// TIA Portal project "Project3" (V17)

(* hardware
DEVICE "S7-1200 station_1"  S7-1200 Station
   slot 0: "Rack_0"  S7-1200 Rack  Rack  V1.0
   slot 1: "PLC_1"  CPU 1212C DC/DC/DC  6ES7 212-1AE40-0XB0  V4.2
DEVICE "HMI_1"  TP700 Comfort
   slot 0: "HMI_1"  TP700 Comfort  6AV2 124-0GC01-0AX0  17.0.0.0
   slot 1: "HMI_RT_1"  TP700 Comfort  6AV2 124-0GC01-0AX0  17.0.0.0
   slot 5: "HMI_1.IE_CP_1"  PROFINET Interface  17.0.0.0
      slot 1: "PROFINET Interface_1"  PROFINET Interface
         slot 1: "Port_1"  Port
         slot 2: "Port_2"  Port
   slot 7: "HMI_1.MPI/DP_CP_1"  MPI/DP Interface  17.0.0.0
*)

// ===== PLC "PLC_1"  CPU 1212C DC/DC/DC =====

VAR_GLOBAL   // PLC tag table "Default tag table"
   "S2" AT %I0.0 : Bool;
   "S3" AT %I0.1 : Bool;
   "S1" AT %I0.2 : Bool;
   "S4" AT %I0.3 : Bool;
   "S5" AT %I0.4 : Bool;
   "Ac" AT %Q0.0 : Bool;
   "Aż" AT %Q0.1 : Bool;
   "Az" AT %Q0.2 : Bool;
   "Bc" AT %Q0.3 : Bool;
   "Bż" AT %Q0.4 : Bool;
   "Bz" AT %Q0.5 : Bool;
   "Clock_Byte" AT %MB100 : Byte;
   "Clock_10Hz" AT %M100.0 : Bool;
   "Clock_5Hz" AT %M100.1 : Bool;
   "Clock_2.5Hz" AT %M100.2 : Bool;
   "Clock_2Hz" AT %M100.3 : Bool;
   "Clock_1.25Hz" AT %M100.4 : Bool;
   "Clock_1Hz" AT %M100.5 : Bool;
   "Clock_0.625Hz" AT %M100.6 : Bool;
   "Clock_0.5Hz" AT %M100.7 : Bool;
   "Start_HMI" AT %M0.0 : Bool;
   "Stop_HMI" AT %M0.1 : Bool;
   "ŻądaniePrzejazdu_HMI" AT %M0.2 : Bool;
   "TrybNocny_HMI" AT %M0.3 : Bool;
   "ResetAwarii_HMI" AT %M0.4 : Bool;
   "Auto/Manual_przycisk" AT %M0.5 : Bool;
   "Ac_HMI" AT %M0.6 : Bool;
   "Aż_HMI" AT %M0.7 : Bool;
   "Az_HMI" AT %M1.0 : Bool;
   "Bc_HMI" AT %M1.1 : Bool;
   "Bż_HMI" AT %M1.2 : Bool;
   "Bz_HMI" AT %M1.3 : Bool;
END_VAR

DATA_BLOCK "Data_block_1"   // DB1
{ S7_Optimized_Access := 'TRUE' }
VERSION : 0.1
   VAR
      ImpulsS4 : Bool;
      TrybNocny : Bool;
      PamiecZboczaS4 : Bool;
      LicznikS4 : Int;
      Awaria : Bool;
      LiczbaCykli : DInt;
      LiczbaPojazdow : DInt;
      LiczbaŻądań : DInt;
      PamiecZboczaS3_2 : Bool;
      PamiecZboczaS3_1 : Bool;
      PamiecZboczaS3 : Bool;
      NumerAktualnegoKroku : Int;
      Pamięć_HMI_Az : Bool;
      Pamięć_HMI_Bz : Bool;
      Pamięć_HMI_Aż : Bool;
      Pamięć_HMI_Bż : Bool;
      Pamięć_HMI_Ac : Bool;
      Pamięć_HMI_Bc : Bool;
      Impuls_HMI_Az : Bool;
      Impuls_HMI_Bz : Bool;
      Impuls_HMI_Aż : Bool;
      Impuls_HMI_Bż : Bool;
      Impuls_HMI_Ac : Bool;
      Impuls_HMI_Bc : Bool;
      Zmiana_Kroku_Wykonana : Bool;
   END_VAR
BEGIN
END_DATA_BLOCK

// folder: System blocks/Program resources

DATA_BLOCK "IEC_Counter_0_DB"   // DB2
{ S7_Optimized_Access := 'TRUE' }
AUTHOR : Simatic
FAMILY : IEC
NAME : CNTR
VERSION : 1.0
// stored: InstanceOfName IEC_COUNTER
"IEC_COUNTER"
BEGIN
END_DATA_BLOCK

DATA_BLOCK "IEC_Timer_0_DB_1"   // DB3
{ S7_Optimized_Access := 'TRUE' }
AUTHOR : Simatic
FAMILY : IEC
NAME : IEC_TMR
VERSION : 1.0
// stored: InstanceOfName IEC_TIMER
"IEC_TIMER"
BEGIN
END_DATA_BLOCK

DATA_BLOCK "IEC_Timer_0_DB_2"   // DB4
{ S7_Optimized_Access := 'TRUE' }
AUTHOR : Simatic
FAMILY : IEC
NAME : IEC_TMR
VERSION : 1.0
// stored: InstanceOfName IEC_TIMER
"IEC_TIMER"
BEGIN
END_DATA_BLOCK

DATA_BLOCK "IEC_Timer_0_DB_3"   // DB5
{ S7_Optimized_Access := 'TRUE' }
AUTHOR : Simatic
FAMILY : IEC
NAME : IEC_TMR
VERSION : 1.0
// stored: InstanceOfName IEC_TIMER
"IEC_TIMER"
BEGIN
END_DATA_BLOCK

DATA_BLOCK "IEC_Timer_0_DB_4"   // DB6
{ S7_Optimized_Access := 'TRUE' }
AUTHOR : Simatic
FAMILY : IEC
NAME : IEC_TMR
VERSION : 1.0
// stored: InstanceOfName IEC_TIMER
"IEC_TIMER"
BEGIN
END_DATA_BLOCK

DATA_BLOCK "IEC_Timer_0_DB_5"   // DB7
{ S7_Optimized_Access := 'TRUE' }
AUTHOR : Simatic
FAMILY : IEC
NAME : IEC_TMR
VERSION : 1.0
// stored: InstanceOfName IEC_TIMER
"IEC_TIMER"
BEGIN
END_DATA_BLOCK

DATA_BLOCK "IEC_Timer_0_DB_6"   // DB8
{ S7_Optimized_Access := 'TRUE' }
AUTHOR : Simatic
FAMILY : IEC
NAME : IEC_TMR
VERSION : 1.0
// stored: InstanceOfName IEC_TIMER
"IEC_TIMER"
BEGIN
END_DATA_BLOCK

DATA_BLOCK "IEC_Timer_0_DB_7"   // DB9
{ S7_Optimized_Access := 'TRUE' }
AUTHOR : Simatic
FAMILY : IEC
NAME : IEC_TMR
VERSION : 1.0
// stored: InstanceOfName IEC_TIMER
"IEC_TIMER"
BEGIN
END_DATA_BLOCK

DATA_BLOCK "IEC_Timer_0_DB_8"   // DB10
{ S7_Optimized_Access := 'TRUE' }
AUTHOR : Simatic
FAMILY : IEC
NAME : IEC_TMR
VERSION : 1.0
// stored: InstanceOfName IEC_TIMER
"IEC_TIMER"
BEGIN
END_DATA_BLOCK

DATA_BLOCK "IEC_Counter_0_DB_1"   // DB11
{ S7_Optimized_Access := 'TRUE' }
AUTHOR : Simatic
FAMILY : IEC
NAME : CNTR
VERSION : 1.0
// stored: InstanceOfName IEC_COUNTER
"IEC_COUNTER"
BEGIN
END_DATA_BLOCK

DATA_BLOCK "IEC_Timer_0_DB"   // DB12
{ S7_Optimized_Access := 'TRUE' }
AUTHOR : Simatic
FAMILY : IEC
NAME : IEC_TMR
VERSION : 1.0
// stored: InstanceOfName IEC_TIMER
"IEC_TIMER"
BEGIN
END_DATA_BLOCK

DATA_BLOCK "IEC_Counter_0_DB_5"   // DB13
{ S7_Optimized_Access := 'TRUE' }
AUTHOR : Simatic
FAMILY : IEC
NAME : CNTR
VERSION : 1.0
// stored: InstanceOfName IEC_COUNTER
"IEC_COUNTER"
BEGIN
END_DATA_BLOCK

DATA_BLOCK "IEC_Timer_0_DB_9"   // DB14
{ S7_Optimized_Access := 'TRUE' }
AUTHOR : Simatic
FAMILY : IEC
NAME : IEC_TMR
VERSION : 1.0
// stored: InstanceOfName IEC_TIMER
"IEC_TIMER"
BEGIN
END_DATA_BLOCK

DATA_BLOCK "IEC_Counter_0_DB_4"   // DB15
{ S7_Optimized_Access := 'TRUE' }
AUTHOR : Simatic
FAMILY : IEC
NAME : CNTR
VERSION : 1.0
// stored: InstanceOfName IEC_COUNTER
"IEC_COUNTER"
BEGIN
END_DATA_BLOCK

DATA_BLOCK "IEC_Timer_0_DB_13"   // DB16
{ S7_Optimized_Access := 'TRUE' }
AUTHOR : Simatic
FAMILY : IEC
NAME : IEC_TMR
VERSION : 1.0
// stored: InstanceOfName IEC_TIMER
"IEC_TIMER"
BEGIN
END_DATA_BLOCK

DATA_BLOCK "IEC_Timer_0_DB_14"   // DB17
{ S7_Optimized_Access := 'TRUE' }
AUTHOR : Simatic
FAMILY : IEC
NAME : IEC_TMR
VERSION : 1.0
// stored: InstanceOfName IEC_TIMER
"IEC_TIMER"
BEGIN
END_DATA_BLOCK

DATA_BLOCK "IEC_Timer_0_DB_15"   // DB18
{ S7_Optimized_Access := 'TRUE' }
AUTHOR : Simatic
FAMILY : IEC
NAME : IEC_TMR
VERSION : 1.0
// stored: InstanceOfName IEC_TIMER
"IEC_TIMER"
BEGIN
END_DATA_BLOCK

DATA_BLOCK "IEC_Timer_0_DB_16"   // DB19
{ S7_Optimized_Access := 'TRUE' }
AUTHOR : Simatic
FAMILY : IEC
NAME : IEC_TMR
VERSION : 1.0
// stored: InstanceOfName IEC_TIMER
"IEC_TIMER"
BEGIN
END_DATA_BLOCK

DATA_BLOCK "IEC_Timer_0_DB_17"   // DB20
{ S7_Optimized_Access := 'TRUE' }
AUTHOR : Simatic
FAMILY : IEC
NAME : IEC_TMR
VERSION : 1.0
// stored: InstanceOfName IEC_TIMER
"IEC_TIMER"
BEGIN
END_DATA_BLOCK

DATA_BLOCK "IEC_Timer_0_DB_18"   // DB21
{ S7_Optimized_Access := 'TRUE' }
AUTHOR : Simatic
FAMILY : IEC
NAME : IEC_TMR
VERSION : 1.0
// stored: InstanceOfName IEC_TIMER
"IEC_TIMER"
BEGIN
END_DATA_BLOCK

DATA_BLOCK "IEC_Timer_0_DB_10"   // DB22
{ S7_Optimized_Access := 'TRUE' }
AUTHOR : Simatic
FAMILY : IEC
NAME : IEC_TMR
VERSION : 1.0
// stored: InstanceOfName IEC_TIMER
"IEC_TIMER"
BEGIN
END_DATA_BLOCK

DATA_BLOCK "IEC_Timer_0_DB_11"   // DB23
{ S7_Optimized_Access := 'TRUE' }
AUTHOR : Simatic
FAMILY : IEC
NAME : IEC_TMR
VERSION : 1.0
// stored: InstanceOfName IEC_TIMER
"IEC_TIMER"
BEGIN
END_DATA_BLOCK

DATA_BLOCK "IEC_Timer_0_DB_12"   // DB24
{ S7_Optimized_Access := 'TRUE' }
AUTHOR : Simatic
FAMILY : IEC
NAME : IEC_TMR
VERSION : 1.0
// stored: InstanceOfName IEC_TIMER
"IEC_TIMER"
BEGIN
END_DATA_BLOCK

// folder: (top level)

ORGANIZATION_BLOCK "Main"   // OB1, LAD, ProgramCycle
TITLE = "Main Program Sweep (Cycle)"
{ S7_Optimized_Access := 'TRUE' }
VERSION : 0.1
   VAR_INPUT
      Initial_Call : Bool;   // Initial call of this OB
      Remanence : Bool;   // =True, if remanent data are available
   END_VAR
   VAR_TEMP   // added for the SCL form of the ladder/FBD networks
      _w1 : Bool;
      _w2 : Bool;
      _w3 : Bool;
      _w4 : Bool;
      _w5 : Bool;
      _w6 : Bool;
   END_VAR
BEGIN

REGION Network 1: Inicjalizacja programu
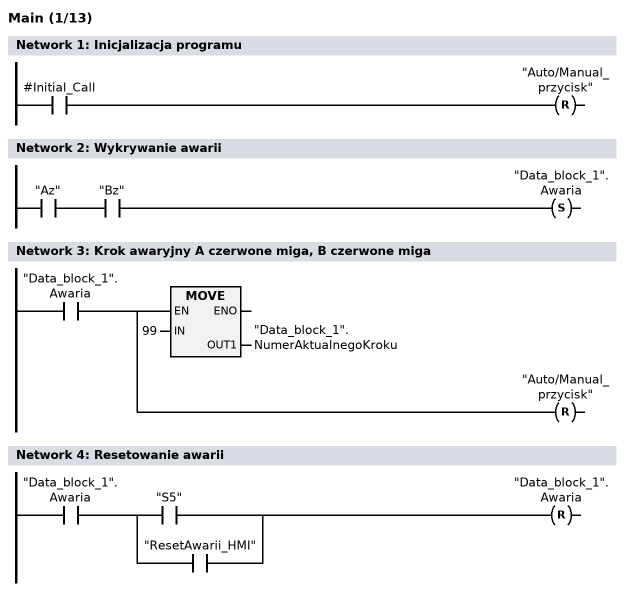
   RUNG wire#powerrail
      Contact( #Initial_Call )
      R_Coil( "Auto/Manual_przycisk" )
   END_RUNG
   // the same network as SCL:
   IF #Initial_Call THEN "Auto/Manual_przycisk" := FALSE; END_IF;
END_REGION

REGION Network 2: Wykrywanie awarii
   RUNG wire#powerrail
      Contact( "Az" )
      Contact( "Bz" )
      S_Coil( "Data_block_1".Awaria )
   END_RUNG
   // the same network as SCL:
   IF "Az" AND "Bz" THEN "Data_block_1".Awaria := TRUE; END_IF;
END_REGION

REGION Network 3: Krok awaryjny A czerwone miga, B czerwone miga
   RUNG wire#powerrail
      Contact( "Data_block_1".Awaria )
      wire#w1
      Move(in := 99, out1 => "Data_block_1".NumerAktualnegoKroku)
   END_RUNG
   RUNG wire#w1
      R_Coil( "Auto/Manual_przycisk" )
   END_RUNG
   // the same network as SCL:
   IF "Data_block_1".Awaria THEN
       "Data_block_1".NumerAktualnegoKroku := 99;
       "Auto/Manual_przycisk" := FALSE;
   END_IF;
END_REGION

REGION Network 4: Resetowanie awarii
   RUNG wire#powerrail
      Contact( "Data_block_1".Awaria )
      wire#w1
      Contact( "S5" )
      wire#w2
      R_Coil( "Data_block_1".Awaria )
   END_RUNG
   RUNG wire#w1
      Contact( "ResetAwarii_HMI" )
   END_RUNG wire#w2
   // the same network as SCL:
   IF "Data_block_1".Awaria AND ("S5" OR "ResetAwarii_HMI") THEN "Data_block_1".Awaria := FALSE; END_IF;
END_REGION

REGION Network 5: Tryb nocny
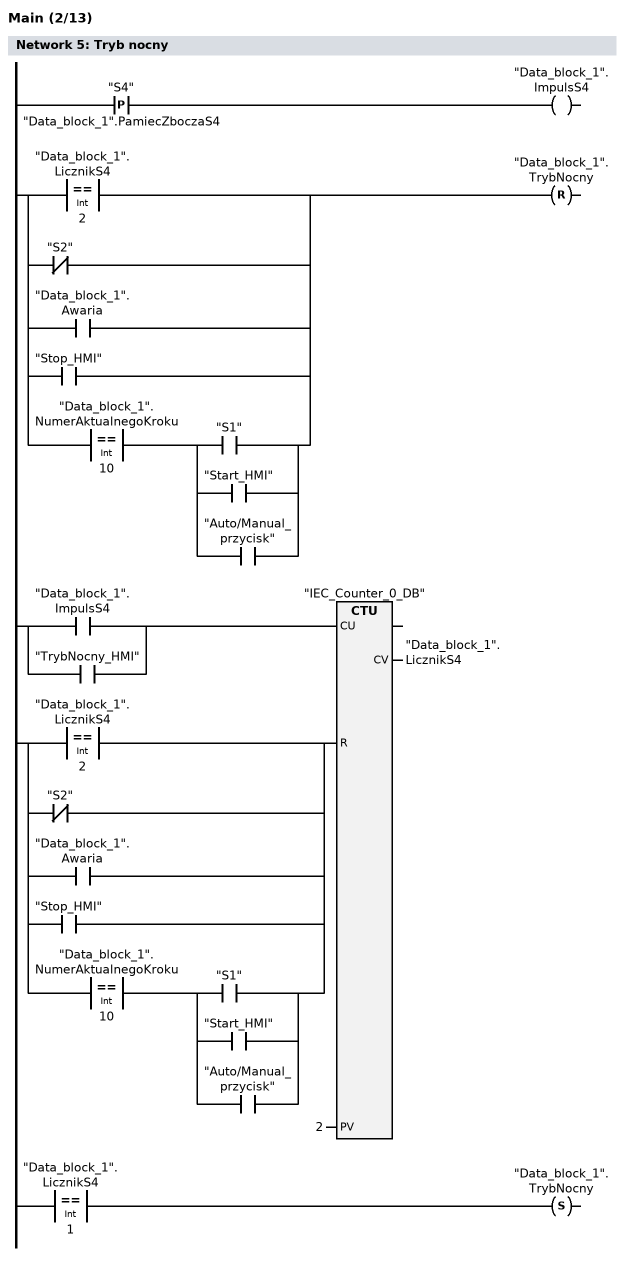
   #_w1 := "S4" AND NOT "Data_block_1".PamiecZboczaS4;   // rising edge of "S4"
   "Data_block_1".PamiecZboczaS4 := "S4";
   "Data_block_1".ImpulsS4 := #_w1;
   IF ("Data_block_1".LicznikS4 = 2) OR NOT "S2" OR "Data_block_1".Awaria OR "Stop_HMI" OR (("Data_block_1".NumerAktualnegoKroku = 10) AND ("S1" OR "Start_HMI" OR "Auto/Manual_przycisk")) THEN
       "Data_block_1".TrybNocny := FALSE;
   END_IF;
   "IEC_Counter_0_DB".CTU(CU := "Data_block_1".ImpulsS4 OR "TrybNocny_HMI",
                          R := ("Data_block_1".LicznikS4 = 2) OR NOT "S2" OR "Data_block_1".Awaria OR "Stop_HMI" OR (("Data_block_1".NumerAktualnegoKroku = 10) AND ("S1" OR "Start_HMI" OR "Auto/Manual_przycisk")),
                          PV := 2,
                          CV => "Data_block_1".LicznikS4);
   IF "Data_block_1".LicznikS4 = 1 THEN "Data_block_1".TrybNocny := TRUE; END_IF;
END_REGION

REGION Network 6: Impulsy HMI
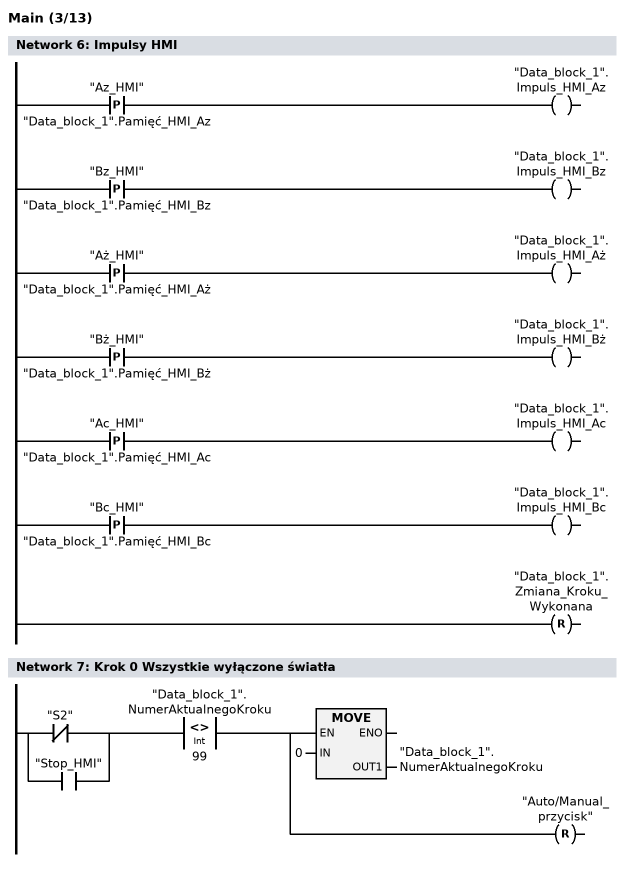
   RUNG wire#powerrail
      P_Contact(operand := "Az_HMI", bit := "Data_block_1".Pamięć_HMI_Az)
      Coil( "Data_block_1".Impuls_HMI_Az )
   END_RUNG
   RUNG wire#powerrail
      P_Contact(operand := "Bz_HMI", bit := "Data_block_1".Pamięć_HMI_Bz)
      Coil( "Data_block_1".Impuls_HMI_Bz )
   END_RUNG
   RUNG wire#powerrail
      P_Contact(operand := "Aż_HMI", bit := "Data_block_1".Pamięć_HMI_Aż)
      Coil( "Data_block_1".Impuls_HMI_Aż )
   END_RUNG
   RUNG wire#powerrail
      P_Contact(operand := "Bż_HMI", bit := "Data_block_1".Pamięć_HMI_Bż)
      Coil( "Data_block_1".Impuls_HMI_Bż )
   END_RUNG
   RUNG wire#powerrail
      P_Contact(operand := "Ac_HMI", bit := "Data_block_1".Pamięć_HMI_Ac)
      Coil( "Data_block_1".Impuls_HMI_Ac )
   END_RUNG
   RUNG wire#powerrail
      P_Contact(operand := "Bc_HMI", bit := "Data_block_1".Pamięć_HMI_Bc)
      Coil( "Data_block_1".Impuls_HMI_Bc )
   END_RUNG
   RUNG wire#powerrail
      R_Coil( "Data_block_1".Zmiana_Kroku_Wykonana )
   END_RUNG
   // the same network as SCL:
   #_w1 := "Az_HMI" AND NOT "Data_block_1".Pamięć_HMI_Az;   // rising edge of "Az_HMI"
   "Data_block_1".Pamięć_HMI_Az := "Az_HMI";
   "Data_block_1".Impuls_HMI_Az := #_w1;
   #_w2 := "Bz_HMI" AND NOT "Data_block_1".Pamięć_HMI_Bz;   // rising edge of "Bz_HMI"
   "Data_block_1".Pamięć_HMI_Bz := "Bz_HMI";
   "Data_block_1".Impuls_HMI_Bz := #_w2;
   #_w3 := "Aż_HMI" AND NOT "Data_block_1".Pamięć_HMI_Aż;   // rising edge of "Aż_HMI"
   "Data_block_1".Pamięć_HMI_Aż := "Aż_HMI";
   "Data_block_1".Impuls_HMI_Aż := #_w3;
   #_w4 := "Bż_HMI" AND NOT "Data_block_1".Pamięć_HMI_Bż;   // rising edge of "Bż_HMI"
   "Data_block_1".Pamięć_HMI_Bż := "Bż_HMI";
   "Data_block_1".Impuls_HMI_Bż := #_w4;
   #_w5 := "Ac_HMI" AND NOT "Data_block_1".Pamięć_HMI_Ac;   // rising edge of "Ac_HMI"
   "Data_block_1".Pamięć_HMI_Ac := "Ac_HMI";
   "Data_block_1".Impuls_HMI_Ac := #_w5;
   #_w6 := "Bc_HMI" AND NOT "Data_block_1".Pamięć_HMI_Bc;   // rising edge of "Bc_HMI"
   "Data_block_1".Pamięć_HMI_Bc := "Bc_HMI";
   "Data_block_1".Impuls_HMI_Bc := #_w6;
   "Data_block_1".Zmiana_Kroku_Wykonana := FALSE;
END_REGION

REGION Network 7: Krok 0 Wszystkie wyłączone światła
   RUNG wire#powerrail
      I_Contact( "S2" )
      wire#w1
      { S7_Templates := "SrcType := Int" } NE_Contact(in1 := "Data_block_1".NumerAktualnegoKroku, in2 := 99)
      wire#w2
      Move(in := 0, out1 => "Data_block_1".NumerAktualnegoKroku)
   END_RUNG
   RUNG wire#powerrail
      Contact( "Stop_HMI" )
   END_RUNG wire#w1
   RUNG wire#w2
      R_Coil( "Auto/Manual_przycisk" )
   END_RUNG
   // the same network as SCL:
   #_w1 := (NOT "S2" OR "Stop_HMI") AND ("Data_block_1".NumerAktualnegoKroku <> 99);
   IF #_w1 THEN
       "Data_block_1".NumerAktualnegoKroku := 0;
       "Auto/Manual_przycisk" := FALSE;
   END_IF;
END_REGION

REGION Network 8: Krok 1 i Licznik Cykli - A zielone, B czerwone
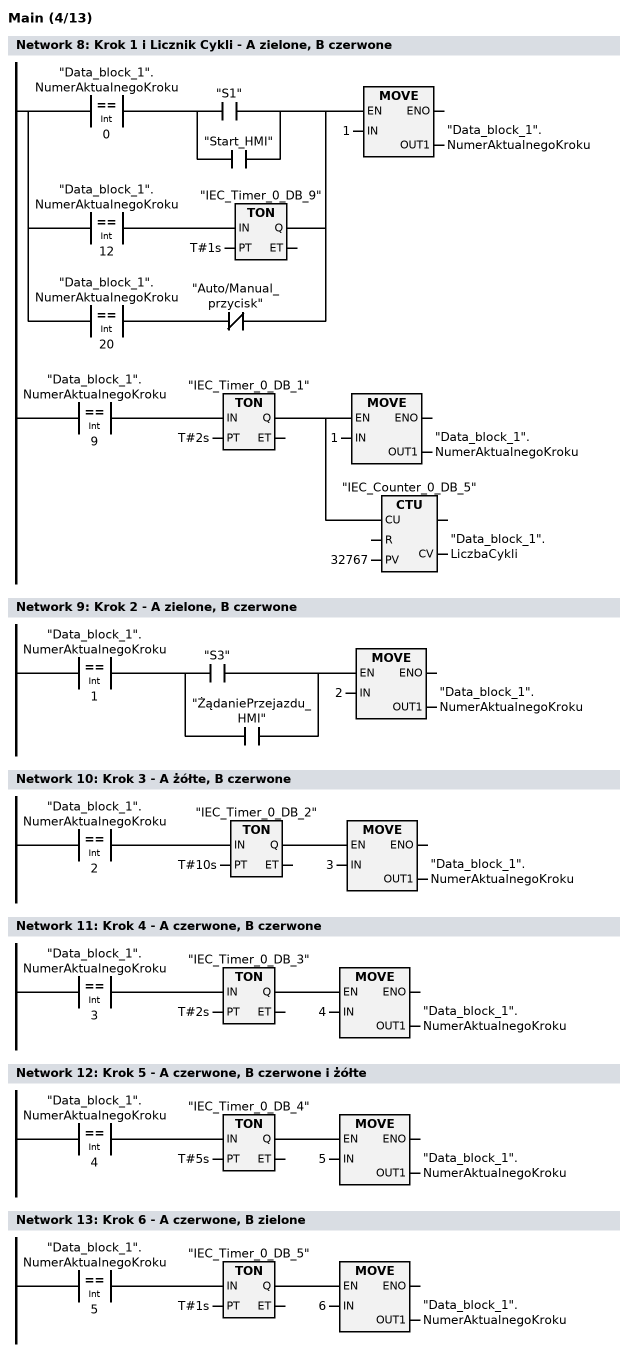
   "IEC_Timer_0_DB_9".TON(IN := "Data_block_1".NumerAktualnegoKroku = 12, PT := T#1s);
   IF (("Data_block_1".NumerAktualnegoKroku = 0) AND ("S1" OR "Start_HMI")) OR "IEC_Timer_0_DB_9".Q OR (("Data_block_1".NumerAktualnegoKroku = 20) AND NOT "Auto/Manual_przycisk") THEN
       "Data_block_1".NumerAktualnegoKroku := 1;
   END_IF;
   "IEC_Timer_0_DB_1".TON(IN := "Data_block_1".NumerAktualnegoKroku = 9, PT := T#2s);
   IF "IEC_Timer_0_DB_1".Q THEN "Data_block_1".NumerAktualnegoKroku := 1; END_IF;
   "IEC_Counter_0_DB_5".CTU(CU := "IEC_Timer_0_DB_1".Q, PV := 32767, CV => "Data_block_1".LiczbaCykli);
END_REGION

REGION Network 9: Krok 2 - A zielone, B czerwone
   RUNG wire#powerrail
      { S7_Templates := "SrcType := Int" } EQ_Contact(in1 := "Data_block_1".NumerAktualnegoKroku, in2 := 1)
      wire#w1
      Contact( "S3" )
      wire#w2
      Move(in := 2, out1 => "Data_block_1".NumerAktualnegoKroku)
   END_RUNG
   RUNG wire#w1
      Contact( "ŻądaniePrzejazdu_HMI" )
   END_RUNG wire#w2
   // the same network as SCL:
   IF ("Data_block_1".NumerAktualnegoKroku = 1) AND ("S3" OR "ŻądaniePrzejazdu_HMI") THEN
       "Data_block_1".NumerAktualnegoKroku := 2;
   END_IF;
END_REGION

REGION Network 10: Krok 3 - A żółte, B czerwone
   "IEC_Timer_0_DB_2".TON(IN := "Data_block_1".NumerAktualnegoKroku = 2, PT := T#10s);
   IF "IEC_Timer_0_DB_2".Q THEN "Data_block_1".NumerAktualnegoKroku := 3; END_IF;
END_REGION

REGION Network 11: Krok 4 - A czerwone, B czerwone
   "IEC_Timer_0_DB_3".TON(IN := "Data_block_1".NumerAktualnegoKroku = 3, PT := T#2s);
   IF "IEC_Timer_0_DB_3".Q THEN "Data_block_1".NumerAktualnegoKroku := 4; END_IF;
END_REGION

REGION Network 12: Krok 5 - A czerwone, B czerwone i żółte
   "IEC_Timer_0_DB_4".TON(IN := "Data_block_1".NumerAktualnegoKroku = 4, PT := T#5s);
   IF "IEC_Timer_0_DB_4".Q THEN "Data_block_1".NumerAktualnegoKroku := 5; END_IF;
END_REGION

REGION Network 13: Krok 6 - A czerwone, B zielone
   "IEC_Timer_0_DB_5".TON(IN := "Data_block_1".NumerAktualnegoKroku = 5, PT := T#1s);
   IF "IEC_Timer_0_DB_5".Q THEN "Data_block_1".NumerAktualnegoKroku := 6; END_IF;
END_REGION

REGION Network 14: Krok 7 - A czerwone, B żółte
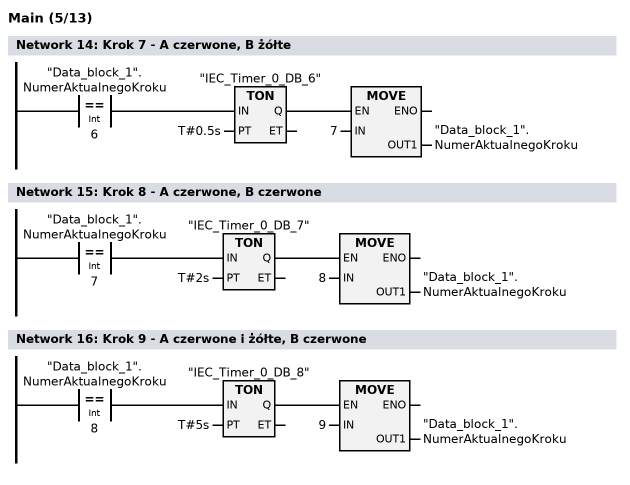
   "IEC_Timer_0_DB_6".TON(IN := "Data_block_1".NumerAktualnegoKroku = 6, PT := T#0.5s);
   IF "IEC_Timer_0_DB_6".Q THEN "Data_block_1".NumerAktualnegoKroku := 7; END_IF;
END_REGION

REGION Network 15: Krok 8 - A czerwone, B czerwone
   "IEC_Timer_0_DB_7".TON(IN := "Data_block_1".NumerAktualnegoKroku = 7, PT := T#2s);
   IF "IEC_Timer_0_DB_7".Q THEN "Data_block_1".NumerAktualnegoKroku := 8; END_IF;
END_REGION

REGION Network 16: Krok 9 - A czerwone i żółte, B czerwone
   "IEC_Timer_0_DB_8".TON(IN := "Data_block_1".NumerAktualnegoKroku = 8, PT := T#5s);
   IF "IEC_Timer_0_DB_8".Q THEN "Data_block_1".NumerAktualnegoKroku := 9; END_IF;
END_REGION

REGION Network 17: Krok 10 - A żółte miga, B żółte miga
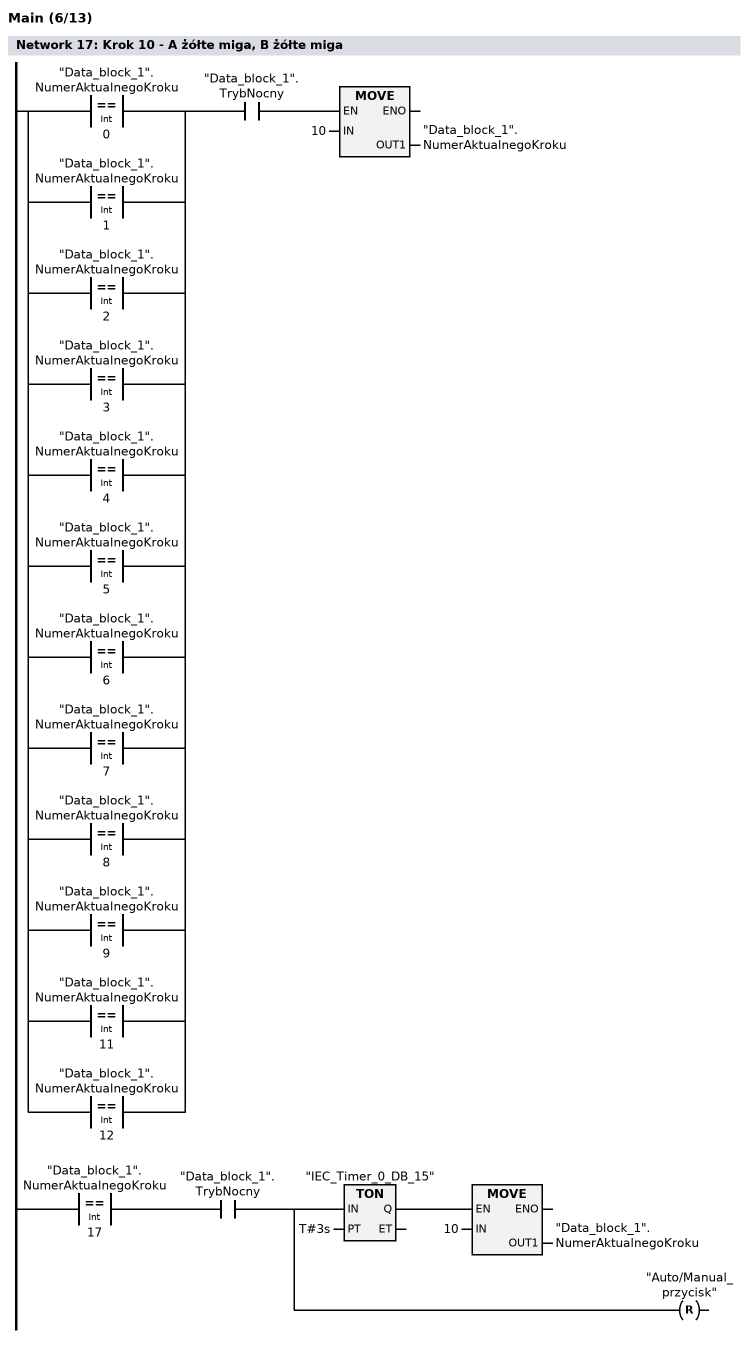
   IF (("Data_block_1".NumerAktualnegoKroku = 0) OR ("Data_block_1".NumerAktualnegoKroku = 1) OR ("Data_block_1".NumerAktualnegoKroku = 2) OR ("Data_block_1".NumerAktualnegoKroku = 3) OR ("Data_block_1".NumerAktualnegoKroku = 4) OR ("Data_block_1".NumerAktualnegoKroku = 5) OR ("Data_block_1".NumerAktualnegoKroku = 6) OR ("Data_block_1".NumerAktualnegoKroku = 7) OR ("Data_block_1".NumerAktualnegoKroku = 8) OR ("Data_block_1".NumerAktualnegoKroku = 9) OR ("Data_block_1".NumerAktualnegoKroku = 11) OR ("Data_block_1".NumerAktualnegoKroku = 12)) AND "Data_block_1".TrybNocny THEN
       "Data_block_1".NumerAktualnegoKroku := 10;
   END_IF;
   #_w1 := ("Data_block_1".NumerAktualnegoKroku = 17) AND "Data_block_1".TrybNocny;
   "IEC_Timer_0_DB_15".TON(IN := #_w1, PT := T#3s);
   IF "IEC_Timer_0_DB_15".Q THEN "Data_block_1".NumerAktualnegoKroku := 10; END_IF;
   IF #_w1 THEN "Auto/Manual_przycisk" := FALSE; END_IF;
END_REGION

REGION Network 18: Krok 11 A czerwone, B czerwone
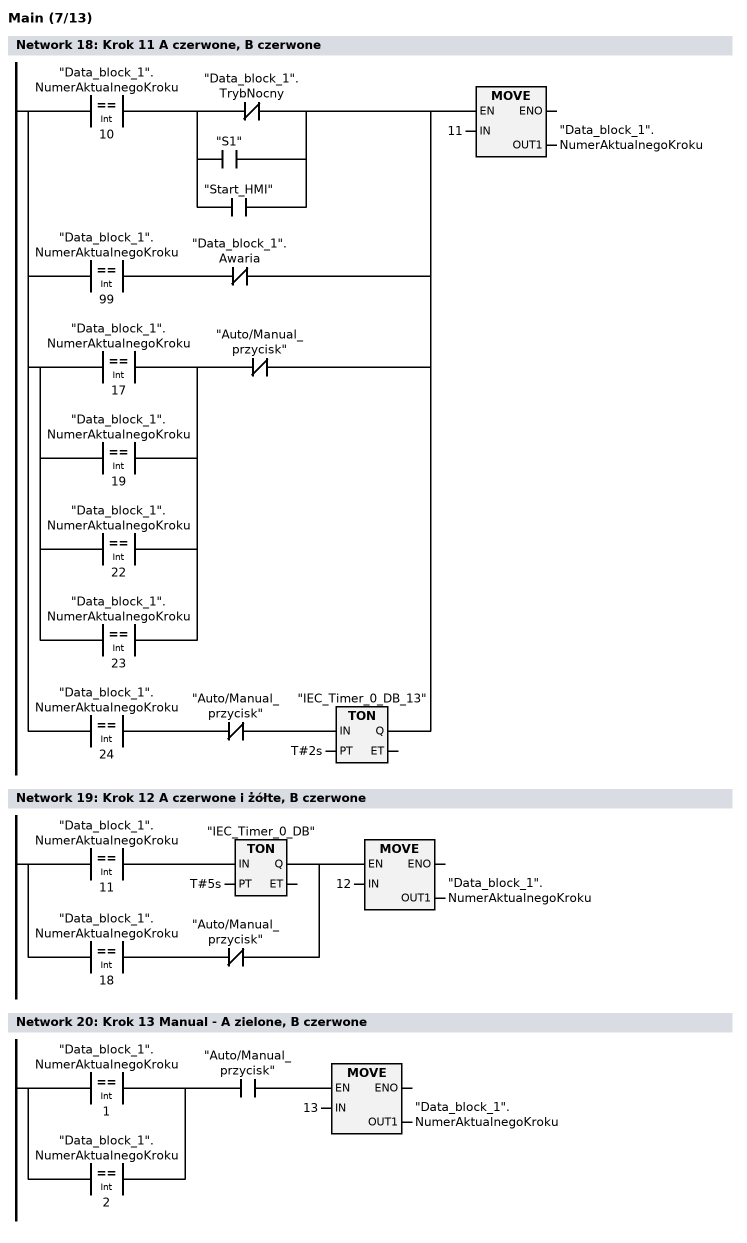
   "IEC_Timer_0_DB_13".TON(IN := ("Data_block_1".NumerAktualnegoKroku = 24) AND NOT "Auto/Manual_przycisk",
                           PT := T#2s);
   IF (("Data_block_1".NumerAktualnegoKroku = 10) AND (NOT "Data_block_1".TrybNocny OR "S1" OR "Start_HMI")) OR (("Data_block_1".NumerAktualnegoKroku = 99) AND NOT "Data_block_1".Awaria) OR ((("Data_block_1".NumerAktualnegoKroku = 17) OR ("Data_block_1".NumerAktualnegoKroku = 19) OR ("Data_block_1".NumerAktualnegoKroku = 22) OR ("Data_block_1".NumerAktualnegoKroku = 23)) AND NOT "Auto/Manual_przycisk") OR "IEC_Timer_0_DB_13".Q THEN
       "Data_block_1".NumerAktualnegoKroku := 11;
   END_IF;
END_REGION

REGION Network 19: Krok 12 A czerwone i żółte, B czerwone
   "IEC_Timer_0_DB".TON(IN := "Data_block_1".NumerAktualnegoKroku = 11, PT := T#5s);
   IF "IEC_Timer_0_DB".Q OR (("Data_block_1".NumerAktualnegoKroku = 18) AND NOT "Auto/Manual_przycisk") THEN
       "Data_block_1".NumerAktualnegoKroku := 12;
   END_IF;
END_REGION

REGION Network 20: Krok 13 Manual - A zielone, B czerwone
   RUNG wire#powerrail
      { S7_Templates := "SrcType := Int" } EQ_Contact(in1 := "Data_block_1".NumerAktualnegoKroku, in2 := 1)
      wire#w1
      Contact( "Auto/Manual_przycisk" )
      Move(in := 13, out1 => "Data_block_1".NumerAktualnegoKroku)
   END_RUNG
   RUNG wire#powerrail
      { S7_Templates := "SrcType := Int" } EQ_Contact(in1 := "Data_block_1".NumerAktualnegoKroku, in2 := 2)
   END_RUNG wire#w1
   // the same network as SCL:
   IF (("Data_block_1".NumerAktualnegoKroku = 1) OR ("Data_block_1".NumerAktualnegoKroku = 2)) AND "Auto/Manual_przycisk" THEN
       "Data_block_1".NumerAktualnegoKroku := 13;
   END_IF;
END_REGION

REGION Network 21: Krok 14 Manual - A żółte, B czerwone
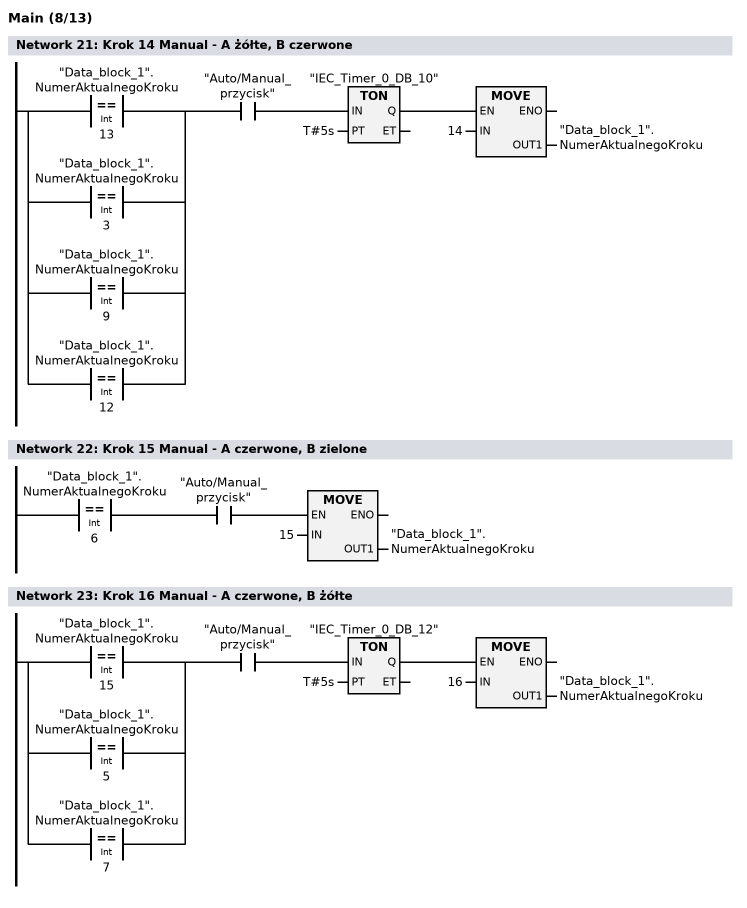
   "IEC_Timer_0_DB_10".TON(IN := (("Data_block_1".NumerAktualnegoKroku = 13) OR ("Data_block_1".NumerAktualnegoKroku = 3) OR ("Data_block_1".NumerAktualnegoKroku = 9) OR ("Data_block_1".NumerAktualnegoKroku = 12)) AND "Auto/Manual_przycisk",
                           PT := T#5s);
   IF "IEC_Timer_0_DB_10".Q THEN "Data_block_1".NumerAktualnegoKroku := 14; END_IF;
END_REGION

REGION Network 22: Krok 15 Manual - A czerwone, B zielone
   RUNG wire#powerrail
      { S7_Templates := "SrcType := Int" } EQ_Contact(in1 := "Data_block_1".NumerAktualnegoKroku, in2 := 6)
      Contact( "Auto/Manual_przycisk" )
      Move(in := 15, out1 => "Data_block_1".NumerAktualnegoKroku)
   END_RUNG
   // the same network as SCL:
   IF ("Data_block_1".NumerAktualnegoKroku = 6) AND "Auto/Manual_przycisk" THEN
       "Data_block_1".NumerAktualnegoKroku := 15;
   END_IF;
END_REGION

REGION Network 23: Krok 16 Manual - A czerwone, B żółte
   "IEC_Timer_0_DB_12".TON(IN := (("Data_block_1".NumerAktualnegoKroku = 15) OR ("Data_block_1".NumerAktualnegoKroku = 5) OR ("Data_block_1".NumerAktualnegoKroku = 7)) AND "Auto/Manual_przycisk",
                           PT := T#5s);
   IF "IEC_Timer_0_DB_12".Q THEN "Data_block_1".NumerAktualnegoKroku := 16; END_IF;
END_REGION

REGION Network 24: Krok 17 Manual - A czerwone, B czerwone
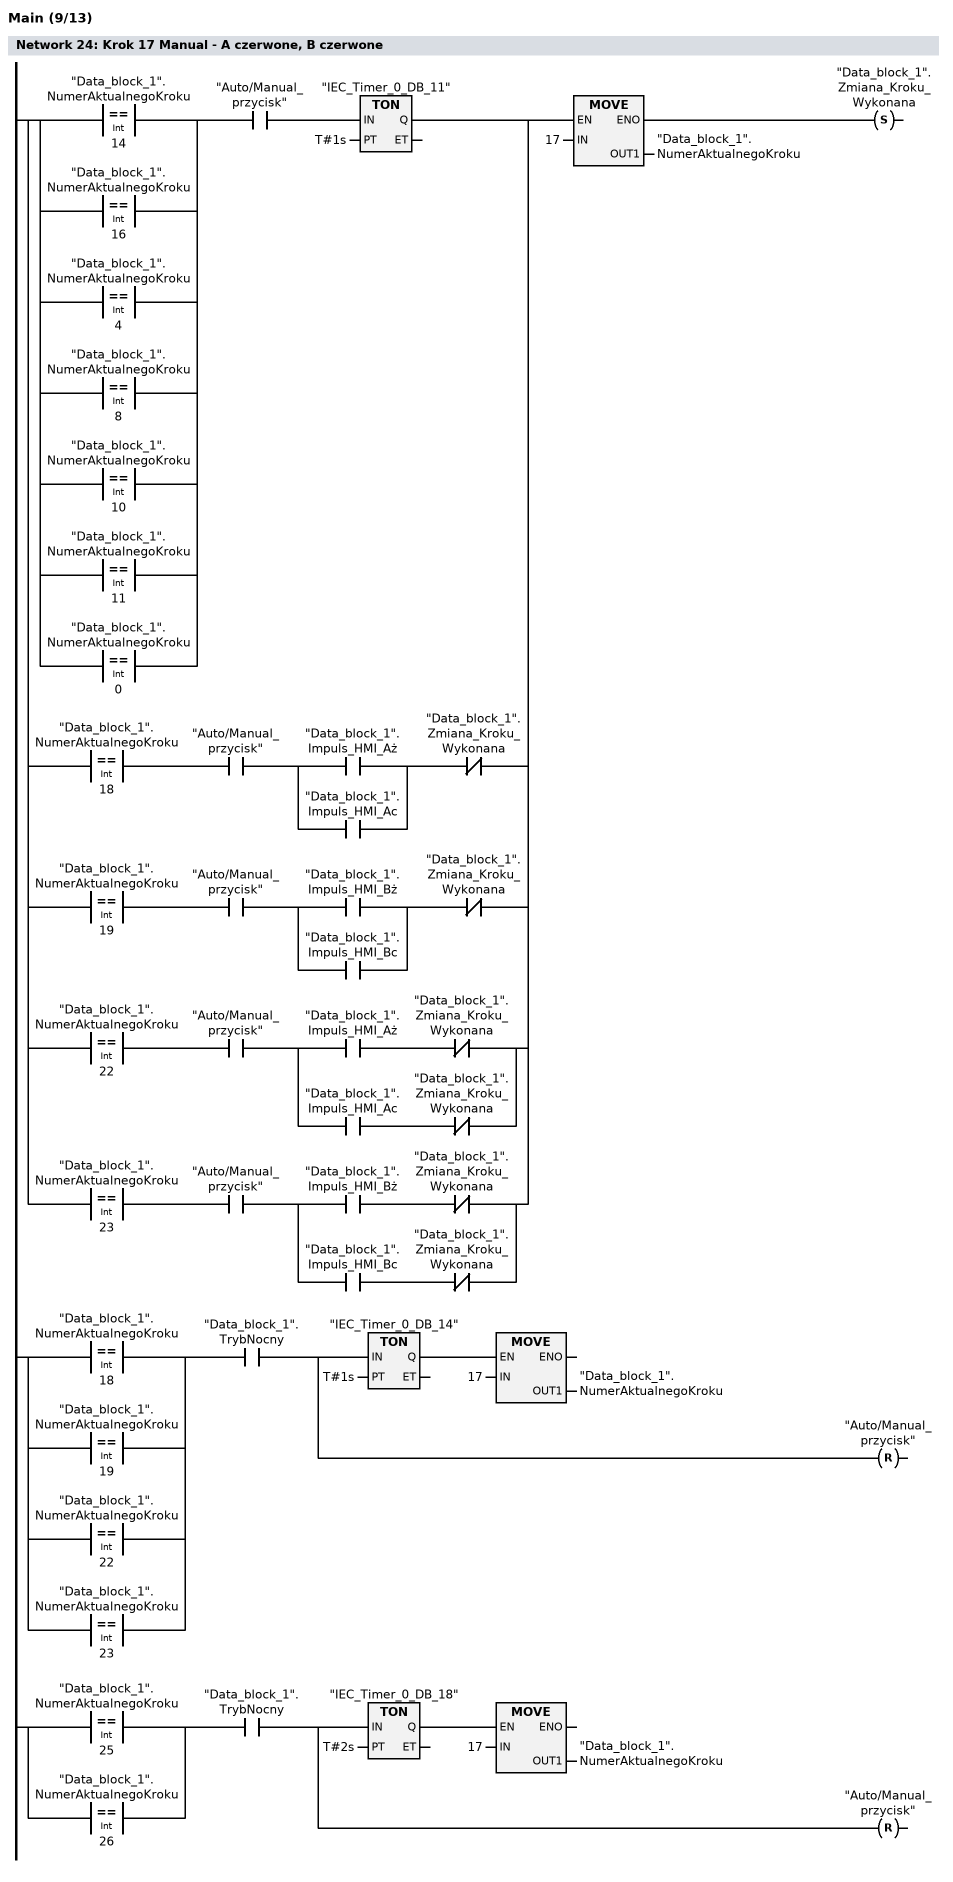
   "IEC_Timer_0_DB_11".TON(IN := (("Data_block_1".NumerAktualnegoKroku = 14) OR ("Data_block_1".NumerAktualnegoKroku = 16) OR ("Data_block_1".NumerAktualnegoKroku = 4) OR ("Data_block_1".NumerAktualnegoKroku = 8) OR ("Data_block_1".NumerAktualnegoKroku = 10) OR ("Data_block_1".NumerAktualnegoKroku = 11) OR ("Data_block_1".NumerAktualnegoKroku = 0)) AND "Auto/Manual_przycisk",
                           PT := T#1s);
   #_w1 := "IEC_Timer_0_DB_11".Q OR (("Data_block_1".NumerAktualnegoKroku = 18) AND "Auto/Manual_przycisk" AND ("Data_block_1".Impuls_HMI_Aż OR "Data_block_1".Impuls_HMI_Ac) AND NOT "Data_block_1".Zmiana_Kroku_Wykonana) OR (("Data_block_1".NumerAktualnegoKroku = 19) AND "Auto/Manual_przycisk" AND ("Data_block_1".Impuls_HMI_Bż OR "Data_block_1".Impuls_HMI_Bc) AND NOT "Data_block_1".Zmiana_Kroku_Wykonana) OR (("Data_block_1".NumerAktualnegoKroku = 22) AND "Auto/Manual_przycisk" AND (("Data_block_1".Impuls_HMI_Aż AND NOT "Data_block_1".Zmiana_Kroku_Wykonana) OR ("Data_block_1".Impuls_HMI_Ac AND NOT "Data_block_1".Zmiana_Kroku_Wykonana))) OR (("Data_block_1".NumerAktualnegoKroku = 23) AND "Auto/Manual_przycisk" AND (("Data_block_1".Impuls_HMI_Bż AND NOT "Data_block_1".Zmiana_Kroku_Wykonana) OR ("Data_block_1".Impuls_HMI_Bc AND NOT "Data_block_1".Zmiana_Kroku_Wykonana)));
   IF #_w1 THEN
       "Data_block_1".NumerAktualnegoKroku := 17;
       "Data_block_1".Zmiana_Kroku_Wykonana := TRUE;
   END_IF;
   #_w2 := (("Data_block_1".NumerAktualnegoKroku = 18) OR ("Data_block_1".NumerAktualnegoKroku = 19) OR ("Data_block_1".NumerAktualnegoKroku = 22) OR ("Data_block_1".NumerAktualnegoKroku = 23)) AND "Data_block_1".TrybNocny;
   "IEC_Timer_0_DB_14".TON(IN := #_w2, PT := T#1s);
   IF "IEC_Timer_0_DB_14".Q THEN "Data_block_1".NumerAktualnegoKroku := 17; END_IF;
   IF #_w2 THEN "Auto/Manual_przycisk" := FALSE; END_IF;
   #_w3 := (("Data_block_1".NumerAktualnegoKroku = 25) OR ("Data_block_1".NumerAktualnegoKroku = 26)) AND "Data_block_1".TrybNocny;
   "IEC_Timer_0_DB_18".TON(IN := #_w3, PT := T#2s);
   IF "IEC_Timer_0_DB_18".Q THEN "Data_block_1".NumerAktualnegoKroku := 17; END_IF;
   IF #_w3 THEN "Auto/Manual_przycisk" := FALSE; END_IF;
END_REGION

REGION Network 25: Krok 18 Manual - A czerwone i żółte, B czerwone
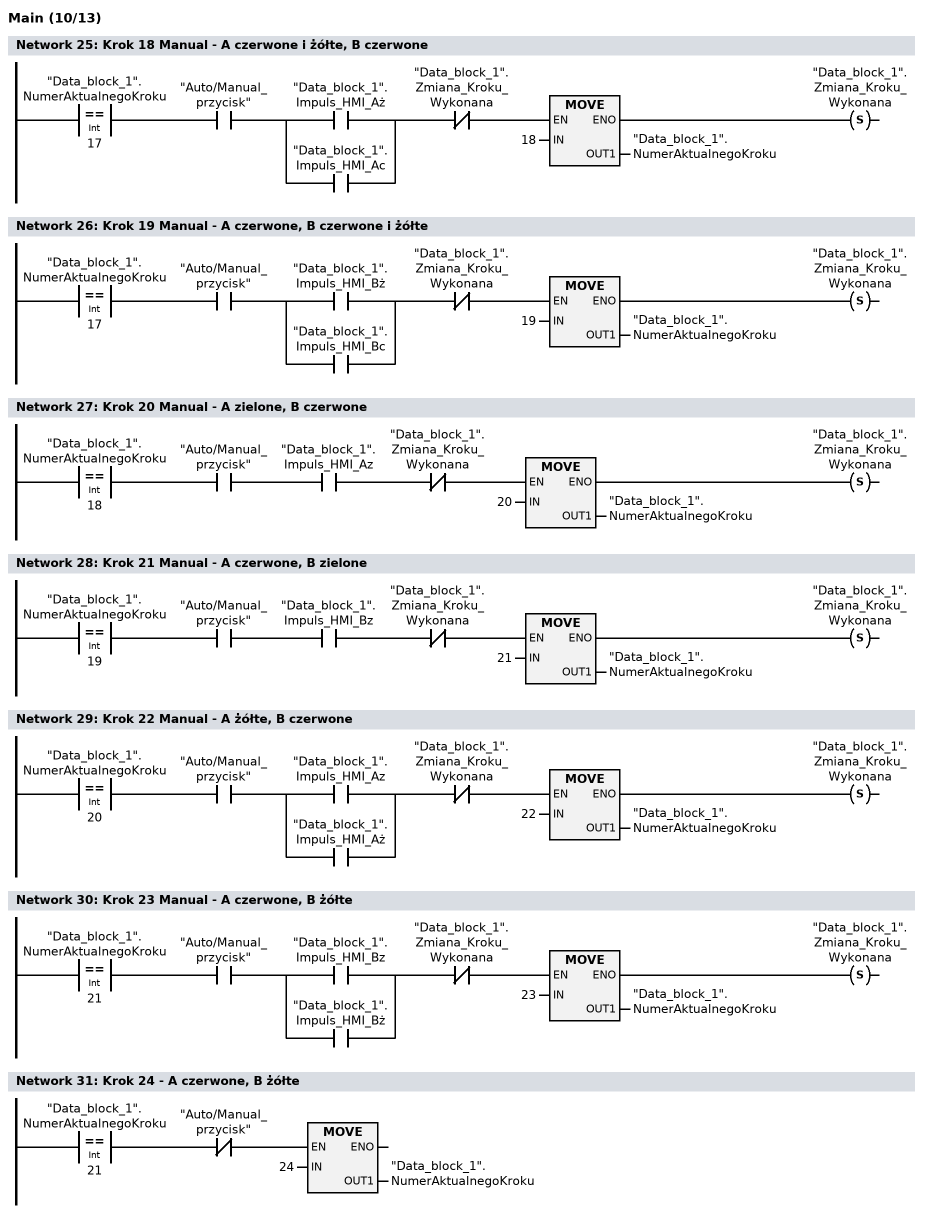
   RUNG wire#powerrail
      { S7_Templates := "SrcType := Int" } EQ_Contact(in1 := "Data_block_1".NumerAktualnegoKroku, in2 := 17)
      Contact( "Auto/Manual_przycisk" )
      wire#w1
      Contact( "Data_block_1".Impuls_HMI_Aż )
      wire#w2
      I_Contact( "Data_block_1".Zmiana_Kroku_Wykonana )
      Move(in := 18, out1 => "Data_block_1".NumerAktualnegoKroku)
      S_Coil( "Data_block_1".Zmiana_Kroku_Wykonana )
   END_RUNG
   RUNG wire#w1
      Contact( "Data_block_1".Impuls_HMI_Ac )
   END_RUNG wire#w2
   // the same network as SCL:
   #_w1 := ("Data_block_1".NumerAktualnegoKroku = 17) AND "Auto/Manual_przycisk" AND ("Data_block_1".Impuls_HMI_Aż OR "Data_block_1".Impuls_HMI_Ac) AND NOT "Data_block_1".Zmiana_Kroku_Wykonana;
   IF #_w1 THEN
       "Data_block_1".NumerAktualnegoKroku := 18;
       "Data_block_1".Zmiana_Kroku_Wykonana := TRUE;
   END_IF;
END_REGION

REGION Network 26: Krok 19 Manual - A czerwone, B czerwone i żółte
   RUNG wire#powerrail
      { S7_Templates := "SrcType := Int" } EQ_Contact(in1 := "Data_block_1".NumerAktualnegoKroku, in2 := 17)
      Contact( "Auto/Manual_przycisk" )
      wire#w1
      Contact( "Data_block_1".Impuls_HMI_Bż )
      wire#w2
      I_Contact( "Data_block_1".Zmiana_Kroku_Wykonana )
      Move(in := 19, out1 => "Data_block_1".NumerAktualnegoKroku)
      S_Coil( "Data_block_1".Zmiana_Kroku_Wykonana )
   END_RUNG
   RUNG wire#w1
      Contact( "Data_block_1".Impuls_HMI_Bc )
   END_RUNG wire#w2
   // the same network as SCL:
   #_w1 := ("Data_block_1".NumerAktualnegoKroku = 17) AND "Auto/Manual_przycisk" AND ("Data_block_1".Impuls_HMI_Bż OR "Data_block_1".Impuls_HMI_Bc) AND NOT "Data_block_1".Zmiana_Kroku_Wykonana;
   IF #_w1 THEN
       "Data_block_1".NumerAktualnegoKroku := 19;
       "Data_block_1".Zmiana_Kroku_Wykonana := TRUE;
   END_IF;
END_REGION

REGION Network 27: Krok 20 Manual - A zielone, B czerwone
   RUNG wire#powerrail
      { S7_Templates := "SrcType := Int" } EQ_Contact(in1 := "Data_block_1".NumerAktualnegoKroku, in2 := 18)
      Contact( "Auto/Manual_przycisk" )
      Contact( "Data_block_1".Impuls_HMI_Az )
      I_Contact( "Data_block_1".Zmiana_Kroku_Wykonana )
      Move(in := 20, out1 => "Data_block_1".NumerAktualnegoKroku)
      S_Coil( "Data_block_1".Zmiana_Kroku_Wykonana )
   END_RUNG
   // the same network as SCL:
   #_w1 := ("Data_block_1".NumerAktualnegoKroku = 18) AND "Auto/Manual_przycisk" AND "Data_block_1".Impuls_HMI_Az AND NOT "Data_block_1".Zmiana_Kroku_Wykonana;
   IF #_w1 THEN
       "Data_block_1".NumerAktualnegoKroku := 20;
       "Data_block_1".Zmiana_Kroku_Wykonana := TRUE;
   END_IF;
END_REGION

REGION Network 28: Krok 21 Manual - A czerwone, B zielone
   RUNG wire#powerrail
      { S7_Templates := "SrcType := Int" } EQ_Contact(in1 := "Data_block_1".NumerAktualnegoKroku, in2 := 19)
      Contact( "Auto/Manual_przycisk" )
      Contact( "Data_block_1".Impuls_HMI_Bz )
      I_Contact( "Data_block_1".Zmiana_Kroku_Wykonana )
      Move(in := 21, out1 => "Data_block_1".NumerAktualnegoKroku)
      S_Coil( "Data_block_1".Zmiana_Kroku_Wykonana )
   END_RUNG
   // the same network as SCL:
   #_w1 := ("Data_block_1".NumerAktualnegoKroku = 19) AND "Auto/Manual_przycisk" AND "Data_block_1".Impuls_HMI_Bz AND NOT "Data_block_1".Zmiana_Kroku_Wykonana;
   IF #_w1 THEN
       "Data_block_1".NumerAktualnegoKroku := 21;
       "Data_block_1".Zmiana_Kroku_Wykonana := TRUE;
   END_IF;
END_REGION

REGION Network 29: Krok 22 Manual - A żółte, B czerwone
   RUNG wire#powerrail
      { S7_Templates := "SrcType := Int" } EQ_Contact(in1 := "Data_block_1".NumerAktualnegoKroku, in2 := 20)
      Contact( "Auto/Manual_przycisk" )
      wire#w1
      Contact( "Data_block_1".Impuls_HMI_Az )
      wire#w2
      I_Contact( "Data_block_1".Zmiana_Kroku_Wykonana )
      Move(in := 22, out1 => "Data_block_1".NumerAktualnegoKroku)
      S_Coil( "Data_block_1".Zmiana_Kroku_Wykonana )
   END_RUNG
   RUNG wire#w1
      Contact( "Data_block_1".Impuls_HMI_Aż )
   END_RUNG wire#w2
   // the same network as SCL:
   #_w1 := ("Data_block_1".NumerAktualnegoKroku = 20) AND "Auto/Manual_przycisk" AND ("Data_block_1".Impuls_HMI_Az OR "Data_block_1".Impuls_HMI_Aż) AND NOT "Data_block_1".Zmiana_Kroku_Wykonana;
   IF #_w1 THEN
       "Data_block_1".NumerAktualnegoKroku := 22;
       "Data_block_1".Zmiana_Kroku_Wykonana := TRUE;
   END_IF;
END_REGION

REGION Network 30: Krok 23 Manual - A czerwone, B żółte
   RUNG wire#powerrail
      { S7_Templates := "SrcType := Int" } EQ_Contact(in1 := "Data_block_1".NumerAktualnegoKroku, in2 := 21)
      Contact( "Auto/Manual_przycisk" )
      wire#w1
      Contact( "Data_block_1".Impuls_HMI_Bz )
      wire#w2
      I_Contact( "Data_block_1".Zmiana_Kroku_Wykonana )
      Move(in := 23, out1 => "Data_block_1".NumerAktualnegoKroku)
      S_Coil( "Data_block_1".Zmiana_Kroku_Wykonana )
   END_RUNG
   RUNG wire#w1
      Contact( "Data_block_1".Impuls_HMI_Bż )
   END_RUNG wire#w2
   // the same network as SCL:
   #_w1 := ("Data_block_1".NumerAktualnegoKroku = 21) AND "Auto/Manual_przycisk" AND ("Data_block_1".Impuls_HMI_Bz OR "Data_block_1".Impuls_HMI_Bż) AND NOT "Data_block_1".Zmiana_Kroku_Wykonana;
   IF #_w1 THEN
       "Data_block_1".NumerAktualnegoKroku := 23;
       "Data_block_1".Zmiana_Kroku_Wykonana := TRUE;
   END_IF;
END_REGION

REGION Network 31: Krok 24 - A czerwone, B żółte
   RUNG wire#powerrail
      { S7_Templates := "SrcType := Int" } EQ_Contact(in1 := "Data_block_1".NumerAktualnegoKroku, in2 := 21)
      I_Contact( "Auto/Manual_przycisk" )
      Move(in := 24, out1 => "Data_block_1".NumerAktualnegoKroku)
   END_RUNG
   // the same network as SCL:
   IF ("Data_block_1".NumerAktualnegoKroku = 21) AND NOT "Auto/Manual_przycisk" THEN
       "Data_block_1".NumerAktualnegoKroku := 24;
   END_IF;
END_REGION

REGION Network 32: Krok 25 - A żółte, B czerwone
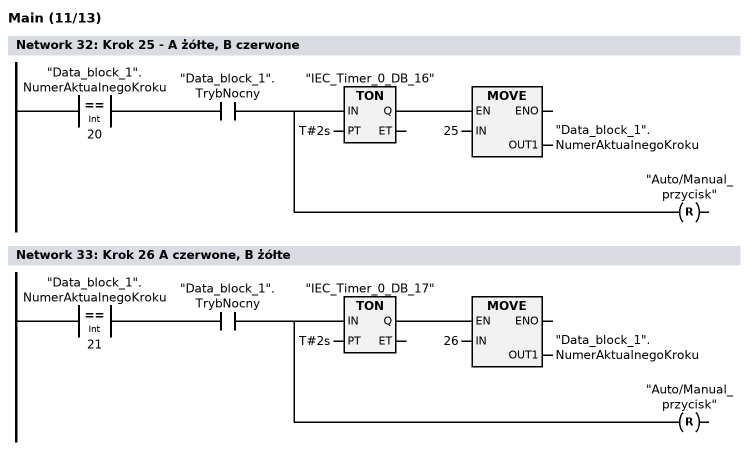
   #_w1 := ("Data_block_1".NumerAktualnegoKroku = 20) AND "Data_block_1".TrybNocny;
   "IEC_Timer_0_DB_16".TON(IN := #_w1, PT := T#2s);
   IF "IEC_Timer_0_DB_16".Q THEN "Data_block_1".NumerAktualnegoKroku := 25; END_IF;
   IF #_w1 THEN "Auto/Manual_przycisk" := FALSE; END_IF;
END_REGION

REGION Network 33: Krok 26 A czerwone, B żółte
   #_w1 := ("Data_block_1".NumerAktualnegoKroku = 21) AND "Data_block_1".TrybNocny;
   "IEC_Timer_0_DB_17".TON(IN := #_w1, PT := T#2s);
   IF "IEC_Timer_0_DB_17".Q THEN "Data_block_1".NumerAktualnegoKroku := 26; END_IF;
   IF #_w1 THEN "Auto/Manual_przycisk" := FALSE; END_IF;
END_REGION

REGION Network 34: Wyjścia
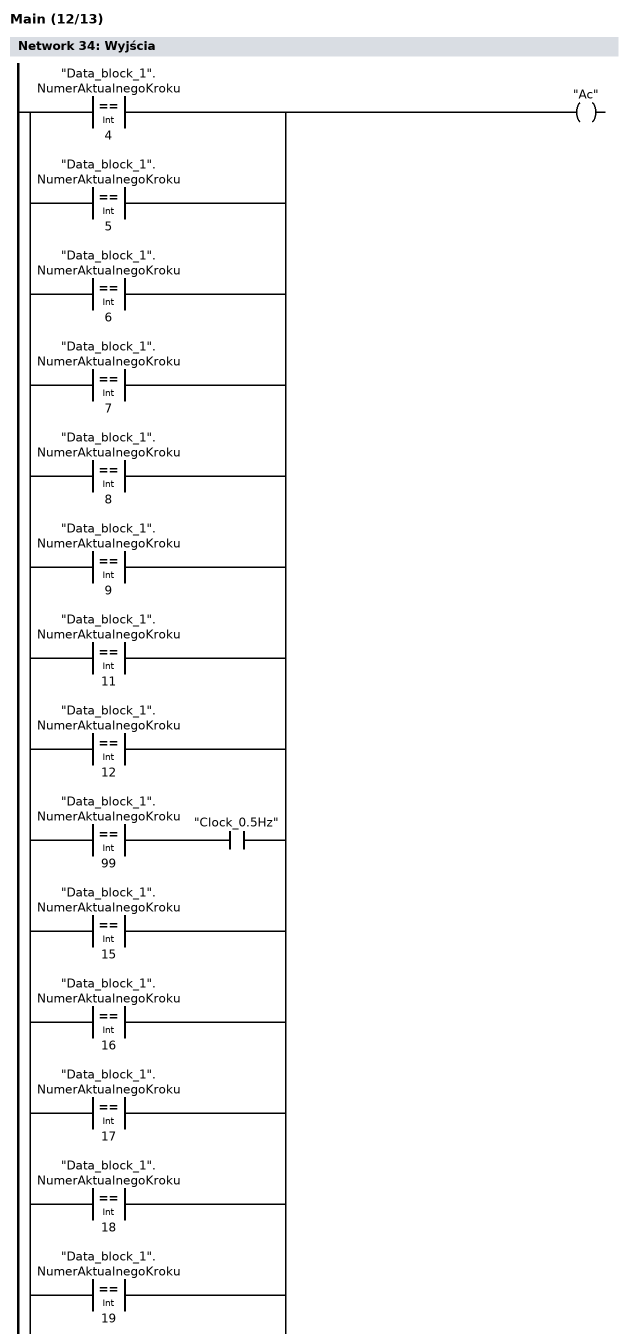
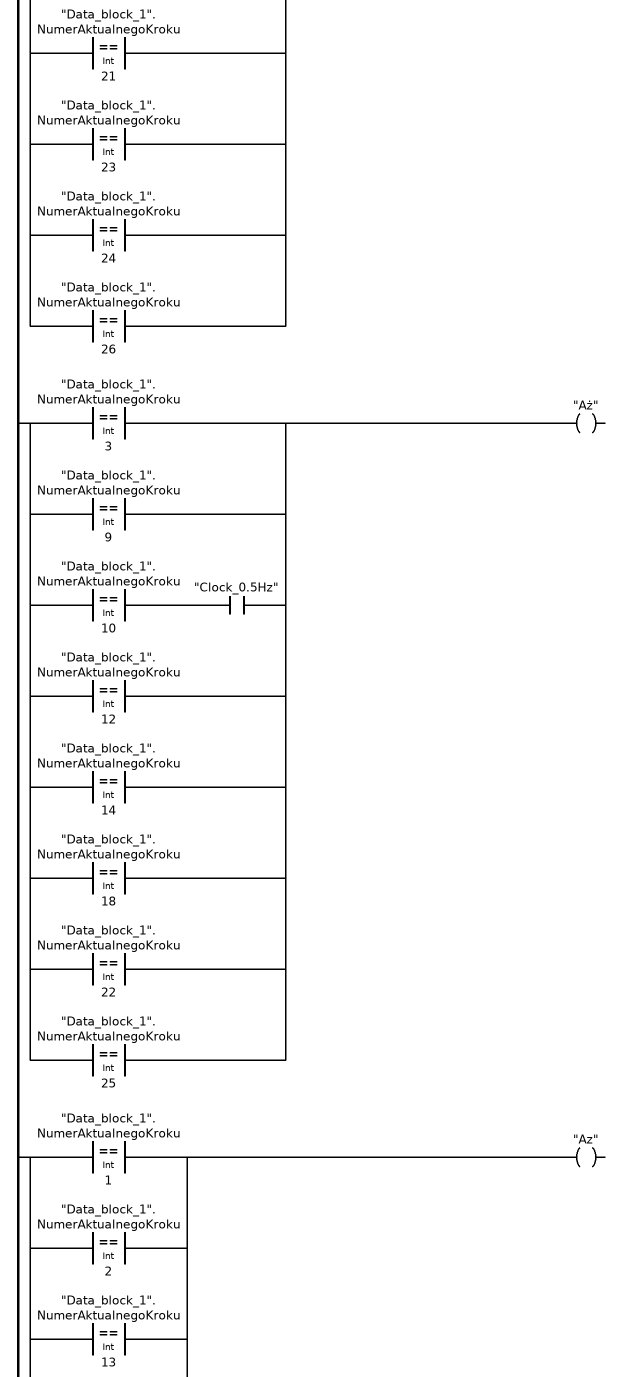
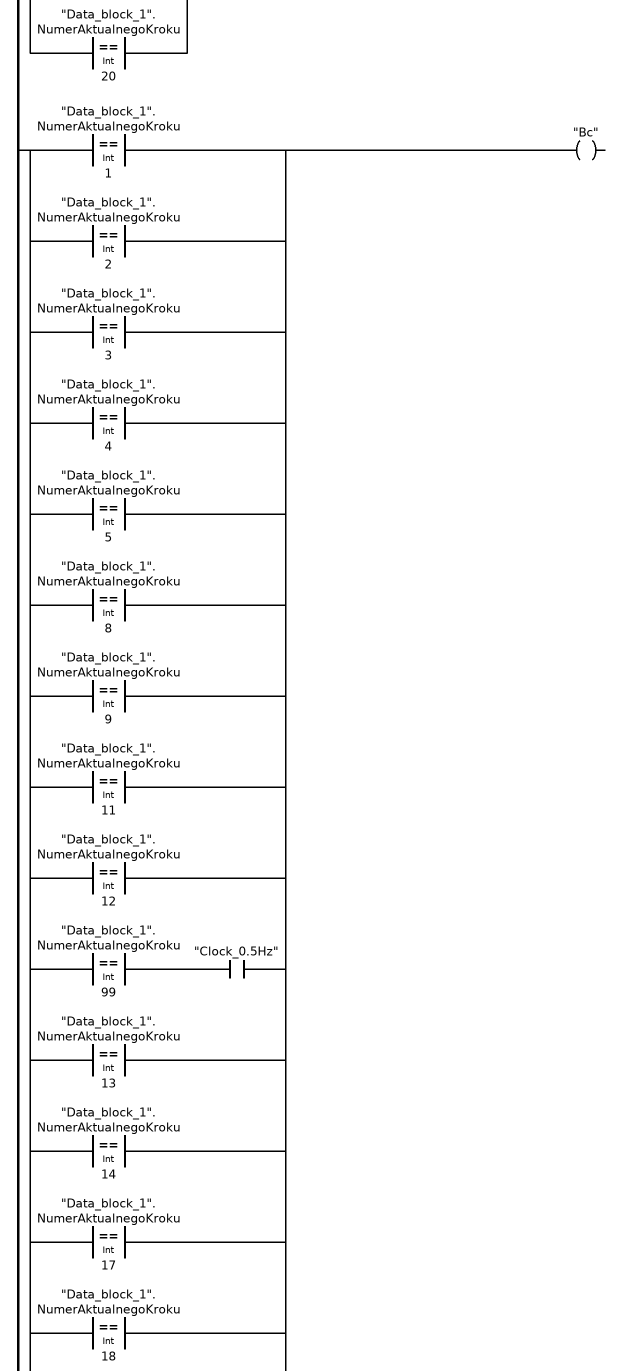
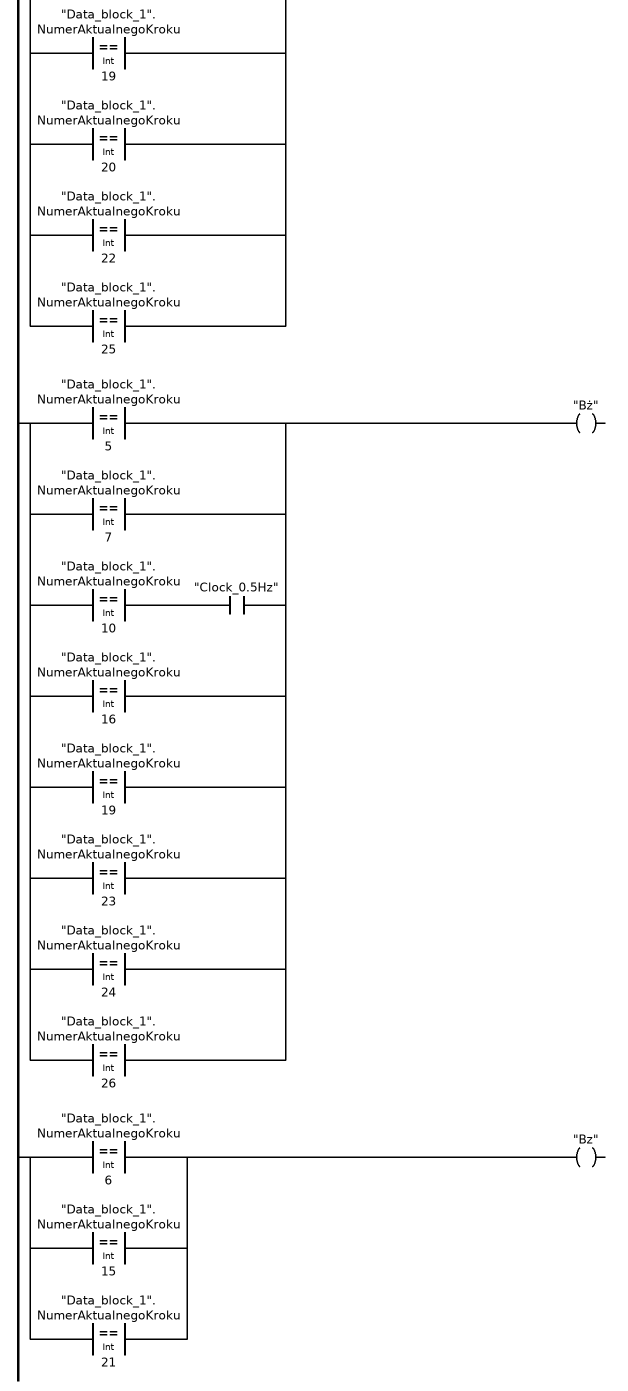
   RUNG wire#powerrail
      { S7_Templates := "SrcType := Int" } EQ_Contact(in1 := "Data_block_1".NumerAktualnegoKroku, in2 := 4)
      wire#w1
      Coil( "Ac" )
   END_RUNG
   RUNG wire#powerrail
      { S7_Templates := "SrcType := Int" } EQ_Contact(in1 := "Data_block_1".NumerAktualnegoKroku, in2 := 5)
   END_RUNG wire#w1
   RUNG wire#powerrail
      { S7_Templates := "SrcType := Int" } EQ_Contact(in1 := "Data_block_1".NumerAktualnegoKroku, in2 := 6)
   END_RUNG wire#w1
   RUNG wire#powerrail
      { S7_Templates := "SrcType := Int" } EQ_Contact(in1 := "Data_block_1".NumerAktualnegoKroku, in2 := 7)
   END_RUNG wire#w1
   RUNG wire#powerrail
      { S7_Templates := "SrcType := Int" } EQ_Contact(in1 := "Data_block_1".NumerAktualnegoKroku, in2 := 8)
   END_RUNG wire#w1
   RUNG wire#powerrail
      { S7_Templates := "SrcType := Int" } EQ_Contact(in1 := "Data_block_1".NumerAktualnegoKroku, in2 := 9)
   END_RUNG wire#w1
   RUNG wire#powerrail
      { S7_Templates := "SrcType := Int" } EQ_Contact(in1 := "Data_block_1".NumerAktualnegoKroku, in2 := 11)
   END_RUNG wire#w1
   RUNG wire#powerrail
      { S7_Templates := "SrcType := Int" } EQ_Contact(in1 := "Data_block_1".NumerAktualnegoKroku, in2 := 12)
   END_RUNG wire#w1
   RUNG wire#powerrail
      { S7_Templates := "SrcType := Int" } EQ_Contact(in1 := "Data_block_1".NumerAktualnegoKroku, in2 := 99)
      Contact( "Clock_0.5Hz" )
   END_RUNG wire#w1
   RUNG wire#powerrail
      { S7_Templates := "SrcType := Int" } EQ_Contact(in1 := "Data_block_1".NumerAktualnegoKroku, in2 := 15)
   END_RUNG wire#w1
   RUNG wire#powerrail
      { S7_Templates := "SrcType := Int" } EQ_Contact(in1 := "Data_block_1".NumerAktualnegoKroku, in2 := 16)
   END_RUNG wire#w1
   RUNG wire#powerrail
      { S7_Templates := "SrcType := Int" } EQ_Contact(in1 := "Data_block_1".NumerAktualnegoKroku, in2 := 17)
   END_RUNG wire#w1
   RUNG wire#powerrail
      { S7_Templates := "SrcType := Int" } EQ_Contact(in1 := "Data_block_1".NumerAktualnegoKroku, in2 := 18)
   END_RUNG wire#w1
   RUNG wire#powerrail
      { S7_Templates := "SrcType := Int" } EQ_Contact(in1 := "Data_block_1".NumerAktualnegoKroku, in2 := 19)
   END_RUNG wire#w1
   RUNG wire#powerrail
      { S7_Templates := "SrcType := Int" } EQ_Contact(in1 := "Data_block_1".NumerAktualnegoKroku, in2 := 21)
   END_RUNG wire#w1
   RUNG wire#powerrail
      { S7_Templates := "SrcType := Int" } EQ_Contact(in1 := "Data_block_1".NumerAktualnegoKroku, in2 := 23)
   END_RUNG wire#w1
   RUNG wire#powerrail
      { S7_Templates := "SrcType := Int" } EQ_Contact(in1 := "Data_block_1".NumerAktualnegoKroku, in2 := 24)
   END_RUNG wire#w1
   RUNG wire#powerrail
      { S7_Templates := "SrcType := Int" } EQ_Contact(in1 := "Data_block_1".NumerAktualnegoKroku, in2 := 26)
   END_RUNG wire#w1
   RUNG wire#powerrail
      { S7_Templates := "SrcType := Int" } EQ_Contact(in1 := "Data_block_1".NumerAktualnegoKroku, in2 := 3)
      wire#w2
      Coil( "Aż" )
   END_RUNG
   RUNG wire#powerrail
      { S7_Templates := "SrcType := Int" } EQ_Contact(in1 := "Data_block_1".NumerAktualnegoKroku, in2 := 9)
   END_RUNG wire#w2
   RUNG wire#powerrail
      { S7_Templates := "SrcType := Int" } EQ_Contact(in1 := "Data_block_1".NumerAktualnegoKroku, in2 := 10)
      Contact( "Clock_0.5Hz" )
   END_RUNG wire#w2
   RUNG wire#powerrail
      { S7_Templates := "SrcType := Int" } EQ_Contact(in1 := "Data_block_1".NumerAktualnegoKroku, in2 := 12)
   END_RUNG wire#w2
   RUNG wire#powerrail
      { S7_Templates := "SrcType := Int" } EQ_Contact(in1 := "Data_block_1".NumerAktualnegoKroku, in2 := 14)
   END_RUNG wire#w2
   RUNG wire#powerrail
      { S7_Templates := "SrcType := Int" } EQ_Contact(in1 := "Data_block_1".NumerAktualnegoKroku, in2 := 18)
   END_RUNG wire#w2
   RUNG wire#powerrail
      { S7_Templates := "SrcType := Int" } EQ_Contact(in1 := "Data_block_1".NumerAktualnegoKroku, in2 := 22)
   END_RUNG wire#w2
   RUNG wire#powerrail
      { S7_Templates := "SrcType := Int" } EQ_Contact(in1 := "Data_block_1".NumerAktualnegoKroku, in2 := 25)
   END_RUNG wire#w2
   RUNG wire#powerrail
      { S7_Templates := "SrcType := Int" } EQ_Contact(in1 := "Data_block_1".NumerAktualnegoKroku, in2 := 1)
      wire#w3
      Coil( "Az" )
   END_RUNG
   RUNG wire#powerrail
      { S7_Templates := "SrcType := Int" } EQ_Contact(in1 := "Data_block_1".NumerAktualnegoKroku, in2 := 2)
   END_RUNG wire#w3
   RUNG wire#powerrail
      { S7_Templates := "SrcType := Int" } EQ_Contact(in1 := "Data_block_1".NumerAktualnegoKroku, in2 := 13)
   END_RUNG wire#w3
   RUNG wire#powerrail
      { S7_Templates := "SrcType := Int" } EQ_Contact(in1 := "Data_block_1".NumerAktualnegoKroku, in2 := 20)
   END_RUNG wire#w3
   RUNG wire#powerrail
      { S7_Templates := "SrcType := Int" } EQ_Contact(in1 := "Data_block_1".NumerAktualnegoKroku, in2 := 1)
      wire#w4
      Coil( "Bc" )
   END_RUNG
   RUNG wire#powerrail
      { S7_Templates := "SrcType := Int" } EQ_Contact(in1 := "Data_block_1".NumerAktualnegoKroku, in2 := 2)
   END_RUNG wire#w4
   RUNG wire#powerrail
      { S7_Templates := "SrcType := Int" } EQ_Contact(in1 := "Data_block_1".NumerAktualnegoKroku, in2 := 3)
   END_RUNG wire#w4
   RUNG wire#powerrail
      { S7_Templates := "SrcType := Int" } EQ_Contact(in1 := "Data_block_1".NumerAktualnegoKroku, in2 := 4)
   END_RUNG wire#w4
   RUNG wire#powerrail
      { S7_Templates := "SrcType := Int" } EQ_Contact(in1 := "Data_block_1".NumerAktualnegoKroku, in2 := 5)
   END_RUNG wire#w4
   RUNG wire#powerrail
      { S7_Templates := "SrcType := Int" } EQ_Contact(in1 := "Data_block_1".NumerAktualnegoKroku, in2 := 8)
   END_RUNG wire#w4
   RUNG wire#powerrail
      { S7_Templates := "SrcType := Int" } EQ_Contact(in1 := "Data_block_1".NumerAktualnegoKroku, in2 := 9)
   END_RUNG wire#w4
   RUNG wire#powerrail
      { S7_Templates := "SrcType := Int" } EQ_Contact(in1 := "Data_block_1".NumerAktualnegoKroku, in2 := 11)
   END_RUNG wire#w4
   RUNG wire#powerrail
      { S7_Templates := "SrcType := Int" } EQ_Contact(in1 := "Data_block_1".NumerAktualnegoKroku, in2 := 12)
   END_RUNG wire#w4
   RUNG wire#powerrail
      { S7_Templates := "SrcType := Int" } EQ_Contact(in1 := "Data_block_1".NumerAktualnegoKroku, in2 := 99)
      Contact( "Clock_0.5Hz" )
   END_RUNG wire#w4
   RUNG wire#powerrail
      { S7_Templates := "SrcType := Int" } EQ_Contact(in1 := "Data_block_1".NumerAktualnegoKroku, in2 := 13)
   END_RUNG wire#w4
   RUNG wire#powerrail
      { S7_Templates := "SrcType := Int" } EQ_Contact(in1 := "Data_block_1".NumerAktualnegoKroku, in2 := 14)
   END_RUNG wire#w4
   RUNG wire#powerrail
      { S7_Templates := "SrcType := Int" } EQ_Contact(in1 := "Data_block_1".NumerAktualnegoKroku, in2 := 17)
   END_RUNG wire#w4
   RUNG wire#powerrail
      { S7_Templates := "SrcType := Int" } EQ_Contact(in1 := "Data_block_1".NumerAktualnegoKroku, in2 := 18)
   END_RUNG wire#w4
   RUNG wire#powerrail
      { S7_Templates := "SrcType := Int" } EQ_Contact(in1 := "Data_block_1".NumerAktualnegoKroku, in2 := 19)
   END_RUNG wire#w4
   RUNG wire#powerrail
      { S7_Templates := "SrcType := Int" } EQ_Contact(in1 := "Data_block_1".NumerAktualnegoKroku, in2 := 20)
   END_RUNG wire#w4
   RUNG wire#powerrail
      { S7_Templates := "SrcType := Int" } EQ_Contact(in1 := "Data_block_1".NumerAktualnegoKroku, in2 := 22)
   END_RUNG wire#w4
   RUNG wire#powerrail
      { S7_Templates := "SrcType := Int" } EQ_Contact(in1 := "Data_block_1".NumerAktualnegoKroku, in2 := 25)
   END_RUNG wire#w4
   RUNG wire#powerrail
      { S7_Templates := "SrcType := Int" } EQ_Contact(in1 := "Data_block_1".NumerAktualnegoKroku, in2 := 5)
      wire#w5
      Coil( "Bż" )
   END_RUNG
   RUNG wire#powerrail
      { S7_Templates := "SrcType := Int" } EQ_Contact(in1 := "Data_block_1".NumerAktualnegoKroku, in2 := 7)
   END_RUNG wire#w5
   RUNG wire#powerrail
      { S7_Templates := "SrcType := Int" } EQ_Contact(in1 := "Data_block_1".NumerAktualnegoKroku, in2 := 10)
      Contact( "Clock_0.5Hz" )
   END_RUNG wire#w5
   RUNG wire#powerrail
      { S7_Templates := "SrcType := Int" } EQ_Contact(in1 := "Data_block_1".NumerAktualnegoKroku, in2 := 16)
   END_RUNG wire#w5
   RUNG wire#powerrail
      { S7_Templates := "SrcType := Int" } EQ_Contact(in1 := "Data_block_1".NumerAktualnegoKroku, in2 := 19)
   END_RUNG wire#w5
   RUNG wire#powerrail
      { S7_Templates := "SrcType := Int" } EQ_Contact(in1 := "Data_block_1".NumerAktualnegoKroku, in2 := 23)
   END_RUNG wire#w5
   RUNG wire#powerrail
      { S7_Templates := "SrcType := Int" } EQ_Contact(in1 := "Data_block_1".NumerAktualnegoKroku, in2 := 24)
   END_RUNG wire#w5
   RUNG wire#powerrail
      { S7_Templates := "SrcType := Int" } EQ_Contact(in1 := "Data_block_1".NumerAktualnegoKroku, in2 := 26)
   END_RUNG wire#w5
   RUNG wire#powerrail
      { S7_Templates := "SrcType := Int" } EQ_Contact(in1 := "Data_block_1".NumerAktualnegoKroku, in2 := 6)
      wire#w6
      Coil( "Bz" )
   END_RUNG
   RUNG wire#powerrail
      { S7_Templates := "SrcType := Int" } EQ_Contact(in1 := "Data_block_1".NumerAktualnegoKroku, in2 := 15)
   END_RUNG wire#w6
   RUNG wire#powerrail
      { S7_Templates := "SrcType := Int" } EQ_Contact(in1 := "Data_block_1".NumerAktualnegoKroku, in2 := 21)
   END_RUNG wire#w6
   // the same network as SCL:
   "Ac" := ("Data_block_1".NumerAktualnegoKroku = 4) OR ("Data_block_1".NumerAktualnegoKroku = 5) OR ("Data_block_1".NumerAktualnegoKroku = 6) OR ("Data_block_1".NumerAktualnegoKroku = 7) OR ("Data_block_1".NumerAktualnegoKroku = 8) OR ("Data_block_1".NumerAktualnegoKroku = 9) OR ("Data_block_1".NumerAktualnegoKroku = 11) OR ("Data_block_1".NumerAktualnegoKroku = 12) OR (("Data_block_1".NumerAktualnegoKroku = 99) AND "Clock_0.5Hz") OR ("Data_block_1".NumerAktualnegoKroku = 15) OR ("Data_block_1".NumerAktualnegoKroku = 16) OR ("Data_block_1".NumerAktualnegoKroku = 17) OR ("Data_block_1".NumerAktualnegoKroku = 18) OR ("Data_block_1".NumerAktualnegoKroku = 19) OR ("Data_block_1".NumerAktualnegoKroku = 21) OR ("Data_block_1".NumerAktualnegoKroku = 23) OR ("Data_block_1".NumerAktualnegoKroku = 24) OR ("Data_block_1".NumerAktualnegoKroku = 26);
   "Aż" := ("Data_block_1".NumerAktualnegoKroku = 3) OR ("Data_block_1".NumerAktualnegoKroku = 9) OR (("Data_block_1".NumerAktualnegoKroku = 10) AND "Clock_0.5Hz") OR ("Data_block_1".NumerAktualnegoKroku = 12) OR ("Data_block_1".NumerAktualnegoKroku = 14) OR ("Data_block_1".NumerAktualnegoKroku = 18) OR ("Data_block_1".NumerAktualnegoKroku = 22) OR ("Data_block_1".NumerAktualnegoKroku = 25);
   "Az" := ("Data_block_1".NumerAktualnegoKroku = 1) OR ("Data_block_1".NumerAktualnegoKroku = 2) OR ("Data_block_1".NumerAktualnegoKroku = 13) OR ("Data_block_1".NumerAktualnegoKroku = 20);
   "Bc" := ("Data_block_1".NumerAktualnegoKroku = 1) OR ("Data_block_1".NumerAktualnegoKroku = 2) OR ("Data_block_1".NumerAktualnegoKroku = 3) OR ("Data_block_1".NumerAktualnegoKroku = 4) OR ("Data_block_1".NumerAktualnegoKroku = 5) OR ("Data_block_1".NumerAktualnegoKroku = 8) OR ("Data_block_1".NumerAktualnegoKroku = 9) OR ("Data_block_1".NumerAktualnegoKroku = 11) OR ("Data_block_1".NumerAktualnegoKroku = 12) OR (("Data_block_1".NumerAktualnegoKroku = 99) AND "Clock_0.5Hz") OR ("Data_block_1".NumerAktualnegoKroku = 13) OR ("Data_block_1".NumerAktualnegoKroku = 14) OR ("Data_block_1".NumerAktualnegoKroku = 17) OR ("Data_block_1".NumerAktualnegoKroku = 18) OR ("Data_block_1".NumerAktualnegoKroku = 19) OR ("Data_block_1".NumerAktualnegoKroku = 20) OR ("Data_block_1".NumerAktualnegoKroku = 22) OR ("Data_block_1".NumerAktualnegoKroku = 25);
   "Bż" := ("Data_block_1".NumerAktualnegoKroku = 5) OR ("Data_block_1".NumerAktualnegoKroku = 7) OR (("Data_block_1".NumerAktualnegoKroku = 10) AND "Clock_0.5Hz") OR ("Data_block_1".NumerAktualnegoKroku = 16) OR ("Data_block_1".NumerAktualnegoKroku = 19) OR ("Data_block_1".NumerAktualnegoKroku = 23) OR ("Data_block_1".NumerAktualnegoKroku = 24) OR ("Data_block_1".NumerAktualnegoKroku = 26);
   "Bz" := ("Data_block_1".NumerAktualnegoKroku = 6) OR ("Data_block_1".NumerAktualnegoKroku = 15) OR ("Data_block_1".NumerAktualnegoKroku = 21);
END_REGION

REGION Network 35: Liczniki
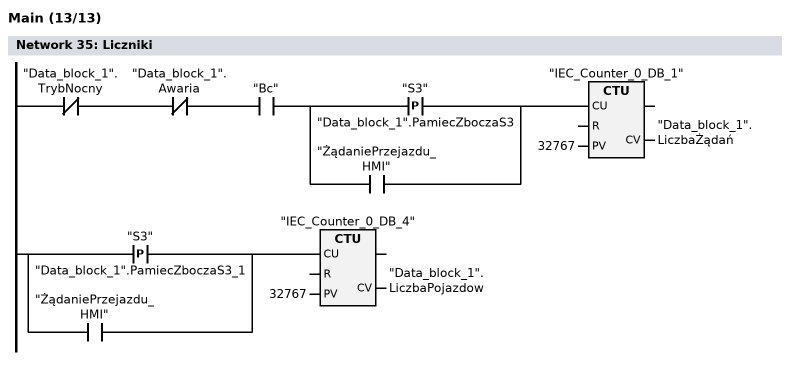
   #_w1 := NOT "Data_block_1".TrybNocny AND NOT "Data_block_1".Awaria AND "Bc" AND "S3" AND NOT "Data_block_1".PamiecZboczaS3;   // rising edge of "S3"
   "Data_block_1".PamiecZboczaS3 := "S3";
   "IEC_Counter_0_DB_1".CTU(CU := #_w1 OR (NOT "Data_block_1".TrybNocny AND NOT "Data_block_1".Awaria AND "Bc" AND "ŻądaniePrzejazdu_HMI"),
                           PV := 32767,
                           CV => "Data_block_1".LiczbaŻądań);
   #_w2 := "S3" AND NOT "Data_block_1".PamiecZboczaS3_1;   // rising edge of "S3"
   "Data_block_1".PamiecZboczaS3_1 := "S3";
   "IEC_Counter_0_DB_4".CTU(CU := #_w2 OR "ŻądaniePrzejazdu_HMI",
                           PV := 32767,
                           CV => "Data_block_1".LiczbaPojazdow);
END_REGION
END_ORGANIZATION_BLOCK

ORGANIZATION_BLOCK "Startup"   // OB100, LAD, Startup
TITLE = "Complete Restart"
{ S7_Optimized_Access := 'TRUE' }
VERSION : 0.1
   VAR_INPUT
      LostRetentive : Bool;   // True if retentive data are lost
      LostRTC : Bool;   // True if date and time are lost
   END_VAR
BEGIN

REGION Network 1
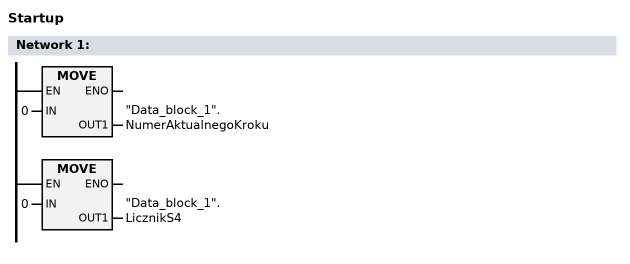
   RUNG wire#powerrail
      Move(in := 0, out1 => "Data_block_1".NumerAktualnegoKroku)
   END_RUNG
   RUNG wire#powerrail
      Move(in := 0, out1 => "Data_block_1".LicznikS4)
   END_RUNG
   // the same network as SCL:
   "Data_block_1".NumerAktualnegoKroku := 0;
   "Data_block_1".LicznikS4 := 0;
END_REGION
END_ORGANIZATION_BLOCK

(* ===== HMI "HMI_RT_1" =====
system functions are stored by id; their names below are inferred from use
connection "HMI_Connection_1": ETHERNET, S7_1200_OMS

HMI tags "Default tag table"
   "Ac" : Bool = PLC Ac AT %Q0.0, 1 s
   "Az" : Bool = PLC Az AT %Q0.2, 1 s
   "Aż" : Bool = PLC Aż AT %Q0.1, 1 s
   "Bc" : Bool = PLC Bc AT %Q0.3, 1 s
   "Bż" : Bool = PLC Bż AT %Q0.4, 1 s
   "Bz" : Bool = PLC Bz AT %Q0.5, 1 s
   "Data_block_1_TrybNocny" : Bool = PLC Data_block_1.TrybNocny, 1 s
   "Data_block_1_Awaria" : Bool = PLC Data_block_1.Awaria, 1 s
   "Data_block_1_LiczbaPojazdow" : DInt = PLC Data_block_1.LiczbaPojazdow, 1 s
   "Data_block_1_LiczbaŻądań" : DInt = PLC Data_block_1.LiczbaŻądań, 1 s
   "Data_block_1_LiczbaCykli" : DInt = PLC Data_block_1.LiczbaCykli, 1 s
   "TrybNocny_HMI" : Bool = PLC TrybNocny_HMI AT %M0.3, 1 s
   "ResetAwarii_HMI" : Bool = PLC ResetAwarii_HMI AT %M0.4, 1 s
   "ŻądaniePrzejazdu_HMI" : Bool = PLC ŻądaniePrzejazdu_HMI AT %M0.2, 1 s
   "Stop_HMI" : Bool = PLC Stop_HMI AT %M0.1, 1 s
   "Start_HMI" : Bool = PLC Start_HMI AT %M0.0, 1 s
   "Data_block_1_NumerAktualnegoKroku" : Int = PLC Data_block_1.NumerAktualnegoKroku, 1 s
   "Auto/Manual_przycisk" : Bool = PLC "Auto/Manual_przycisk" AT %M0.5, 1 s
   "Ac_HMI" : Bool = PLC Ac_HMI AT %M0.6, 1 s
   "Aż_HMI" : Bool = PLC Aż_HMI AT %M0.7, 1 s
   "Az_HMI" : Bool = PLC Az_HMI AT %M1.0, 1 s
   "Bc_HMI" : Bool = PLC Bc_HMI AT %M1.1, 1 s
   "Bż_HMI" : Bool = PLC Bż_HMI AT %M1.2, 1 s
   "Bz_HMI" : Bool = PLC Bz_HMI AT %M1.3, 1 s

screen "Screen_1" 800x480
   Circle "Circle_1" at 97,81 size 48x48
      Appearance <- "Ac"
   TextField "Text field_1" at 52,40 size 149x23; Text 'Skrzyżowanie A'
   TextField "Text field_2" at 261,40 size 148x23; Text 'Skrzyżowanie B'
   Circle "Circle_2" at 97,136 size 48x48
      Appearance <- "Aż"
   Circle "Circle_3" at 97,192 size 48x48
      Appearance <- "Az"
   Circle "Circle_4" at 309,81 size 48x48
      Appearance <- "Bc"
   Circle "Circle_5" at 309,136 size 48x48
      Appearance <- "Bż"
   Circle "Circle_6" at 309,192 size 48x48
      Appearance <- "Bz"
   TextField "Text field_3" at 239,300 size 106x23; Text 'Tryb Nocny'
   TextField "Text field_4" at 257,387 size 69x23; Text 'Awaria'
   Circle "Circle_7" at 264,323 size 48x48
      Appearance <- "Data_block_1_TrybNocny"
   Circle "Circle_8" at 264,410 size 48x48
      Appearance <- "Data_block_1_Awaria"
   TextField "Text field_5" at 62,284 size 161x23; Text 'Licznik pojazdów'
   TextField "Text field_6" at 77,349 size 128x23; Text 'Licznik żądań'
   TextField "Text field_7" at 85,412 size 116x23; Text 'Licznik cykli'
   IOField "I/O field_1" at 89,307 size 96x32; FormatPattern s9999999999
      ProcessValue <- "Data_block_1_LiczbaPojazdow"
   IOField "I/O field_2" at 89,372 size 96x32; FormatPattern s9999999999
      ProcessValue <- "Data_block_1_LiczbaŻądań"
   IOField "I/O field_3" at 89,435 size 96x32; FormatPattern s9999999999
      ProcessValue <- "Data_block_1_LiczbaCykli"
   Button "Button_1" at 578,43 size 96x32; TextOff 'Start'
      on Press: SetBit("Start_HMI")
      on Release: ResetBit("Start_HMI")
   Button "Button_2" at 326,419 size 112x32; TextOff 'Reset awarii'
      on Press: SetBit("ResetAwarii_HMI")
      on Release: ResetBit("ResetAwarii_HMI")
   Button "Button_3" at 578,91 size 96x32; TextOff 'Stop'
      on Press: SetBit("Stop_HMI")
      on Release: ResetBit("Stop_HMI")
   Button "Button_4" at 549,136 size 158x32; TextOff 'Żądanie przejazdu'
      on Press: SetBit("ŻądaniePrzejazdu_HMI")
      on Release: ResetBit("ŻądaniePrzejazdu_HMI")
   Button "Button_5" at 326,329 size 96x32; TextOff 'Tryb Nocny'
      on Press: SetBit("TrybNocny_HMI")
      on Release: ResetBit("TrybNocny_HMI")
   TextField "Text field_8" at 567,403 size 233x23; Text 'Numer Aktualnego Kroku'
   IOField "I/O field_4" at 625,426 size 96x32; FormatPattern s99999
      ProcessValue <- "Data_block_1_NumerAktualnegoKroku"
   Switch "Switch_1" at 568,175 size 120x88; CaptionText 'Manual/Auto'; TextOff 'Auto'; TextOn 'Manual'
      ProcessValue <- "Auto/Manual_przycisk"
   Button "Button_6" at 155,89 size 96x32; TextOff 'Czerwone'
      on Press: SetBit("Ac_HMI")
      on Release: ResetBit("Ac_HMI")
      Visibility <- "Auto/Manual_przycisk"
   Button "Button_7" at 370,89 size 96x32; TextOff 'Czerwone'
      on Press: SetBit("Bc_HMI")
      on Release: ResetBit("Bc_HMI")
      Visibility <- "Auto/Manual_przycisk"
   Button "Button_8" at 155,143 size 96x32; TextOff 'Żółte'
      on Press: SetBit("Aż_HMI")
      on Release: ResetBit("Aż_HMI")
      Visibility <- "Auto/Manual_przycisk"
   Button "Button_9" at 155,199 size 96x32; TextOff 'Zielone'
      on Press: SetBit("Az_HMI")
      on Release: ResetBit("Az_HMI")
      Visibility <- "Auto/Manual_przycisk"
   Button "Button_10" at 370,143 size 96x32; TextOff 'Żółte'
      on Press: SetBit("Bż_HMI")
      on Release: ResetBit("Bż_HMI")
      Visibility <- "Auto/Manual_przycisk"
   Button "Button_11" at 370,199 size 96x32; TextOff 'Zielone'
      on Press: SetBit("Bz_HMI")
      on Release: ResetBit("Bz_HMI")
      Visibility <- "Auto/Manual_przycisk"
*)